// TIA Portal project "Mill3" (V17)

(* hardware
DEVICE "S7-1500/ET200MP station_1"  S7-1500 station
   slot 0: "Rail_0"  Rack  6ES7 590-1***0-0AA0
   slot 1: "PLC_1"  CPU 1512C-1 PN  6ES7 512-1CK01-0AB0  V2.9
      slot 3: "CPU display_1"  6ES7591-1AA00-0AA0
      slot 32768: "PROFINET interface_1"  X1
         slot 32769: "Port_1"  X1 P1
         slot 32770: "Port_2"  X1 P2
      slot 34817: "Virtual CP interface port_1"  Virtual CP interface port  Virtual CP interface port
*)

// ===== PLC "PLC_1"  CPU 1512C-1 PN =====

VAR_GLOBAL   // PLC tag table "Default tag table"
   "Tag_1" AT %M0.0 : Bool;
   "Tag_2" AT %M0.1 : Bool;
   "ResetPID" AT %I0.2 : Bool;
END_VAR

TYPE "Weigh_Feeder"
   STRUCT
      LoadCell_Reading : Real;
      Motor_Speed : Real;
      "SetPoint_%" : Real;
      SetPoint : Real;
      "Maximum_t/h" : Real;
   END_STRUCT;
END_TYPE

TYPE "Motors"
   STRUCT
      Start : Bool;
      Stop : Bool;
      "Motor_ON/OFF" : Bool;
   END_STRUCT;
END_TYPE

TYPE "Belts&BE"
   STRUCT
      Start : Bool;
      Stop : Bool;
      "Belt_ON/OFF" : Bool;
      BSS : Bool;
      PC : Bool;
      PC_Error : Bool;
      BSS_Error : Bool;
      Reset_Error : Bool;
   END_STRUCT;
END_TYPE

TYPE "Ratios"
   STRUCT
      Clinker : Real;
      Pozzolana : Real;
      Gypsum : Real;
      Limestone : Real;
      Select : Bool;
      Selected : Bool;
   END_STRUCT;
END_TYPE

TYPE "bagfilter"
   STRUCT
      Start : Bool;
      Stop : Bool;
      "On/Off" : Bool;
   END_STRUCT;
END_TYPE

TYPE "Reverse/Foward"
   STRUCT
      Foward : Bool;
      Reverse : Bool;
      Stop : Bool;
      PC : Bool;
      BSS : Bool;
      PC_Error : Bool;
      BSS_Error : Bool;
      Reset_Error : Bool;
      FWD_Mode : Bool;
      REV_Mode : Bool;
   END_STRUCT;
END_TYPE

// folder: DataBlocks

DATA_BLOCK "WeighFeeders(DB)"   // DB1
{ S7_Optimized_Access := 'TRUE' }
VERSION : 0.1
   VAR
      Pozzolana : "Weigh_Feeder";
      Clinker : "Weigh_Feeder";
      Gypsum : "Weigh_Feeder";
      Limestone : "Weigh_Feeder";
      Mill_TPH : Real := 310.0;
   END_VAR
BEGIN
   Pozzolana."Maximum_t/h" := 175.0;
   Clinker."Maximum_t/h" := 310.0;
   Gypsum."Maximum_t/h" := 35.0;
   Limestone."Maximum_t/h" := 75.0;
END_DATA_BLOCK

DATA_BLOCK "StartSystem"   // DB6
{ S7_Optimized_Access := 'TRUE' }
VERSION : 0.1
   VAR
      StartSystem : Bool;
      StopSystem : Bool;
      "Syste_ON/OFF" : Bool;
      Automatic_Selection : Bool;
      Manual_Selection : Bool;
      AuromaticMode : Bool;
      ManualMode : Bool;
      Siren : Bool;
      Main_BagFilter : "bagfilter";
      Mill_Drive : "Motors";
      "280KW FAN" : "Motors";
      MainBF_RotorAirLock : "Motors";
      Silo_Level : Int;
      Mill_Temp : Real := 23.0;
      level_Indication : Int;
      Timer1_PT : Time := T#15000ms;
      Timer2_PT : Time := T#10000ms;
   END_VAR
BEGIN
END_DATA_BLOCK

DATA_BLOCK "Belts|BE"   // DB9
{ S7_Optimized_Access := 'TRUE' }
VERSION : 0.1
   VAR
      Clinker : "Belts&BE";
      Pozzolana : "Belts&BE";
      Gypsum : "Belts&BE";
      Limestone : "Belts&BE";
      MaterialInlet_Belt : "Belts&BE";
      CourseMaterial_Belt : "Belts&BE";
      MillInlet_BE : "Belts&BE";
      OutletSilo_BE : "Belts&BE";
      FromYard_Belt : "Belts&BE";
      BF_To_OutletBE_Belt : "Belts&BE";
      "Clinker&Gypsum_Belt" : "Reverse/Foward";
      "Limestone&Pozzolana_Belt" : "Reverse/Foward";
   END_VAR
BEGIN
END_DATA_BLOCK

DATA_BLOCK "Material Rationing"   // DB10
{ S7_Optimized_Access := 'TRUE' }
VERSION : 0.1
   VAR
      Kp_Silver : "Ratios";
      Kp_Gold : "Ratios";
      Kp_Super_Gold : "Ratios";
      Kp_OPC : "Ratios";
   END_VAR
BEGIN
   Kp_Silver.Clinker := 52.0;
   Kp_Silver.Pozzolana := 40.0;
   Kp_Silver.Gypsum := 3.0;
   Kp_Silver.Limestone := 5.0;
   Kp_OPC.Clinker := 92.0;
   Kp_OPC.Pozzolana := 0.0;
   Kp_OPC.Gypsum := 5.0;
   Kp_OPC.Limestone := 3.0;
   Kp_Super_Gold.Clinker := 80.0;
   Kp_Super_Gold.Pozzolana := 10.0;
   Kp_Super_Gold.Gypsum := 5.0;
   Kp_Super_Gold.Limestone := 5.0;
   Kp_Gold.Clinker := 72.0;
   Kp_Gold.Pozzolana := 20.0;
   Kp_Gold.Gypsum := 5.0;
   Kp_Gold.Limestone := 3.0;
END_DATA_BLOCK

// folder: System blocks/Program resources

DATA_BLOCK "IEC_Timer_0_DB"   // DB7
{ S7_Optimized_Access := 'TRUE' }
AUTHOR : Simatic
FAMILY : IEC
NAME : IEC_TMR
VERSION : 1.0
// stored: InstanceOfName IEC_TIMER
"IEC_TIMER"
BEGIN
END_DATA_BLOCK

DATA_BLOCK "IEC_Timer_0_DB_1"   // DB8
{ S7_Optimized_Access := 'TRUE' }
AUTHOR : Simatic
FAMILY : IEC
NAME : IEC_TMR
VERSION : 1.0
// stored: InstanceOfName IEC_TIMER
"IEC_TIMER"
BEGIN
END_DATA_BLOCK

// folder: (top level)

ORGANIZATION_BLOCK "Main"   // OB1, LAD, ProgramCycle
TITLE = "Main Program Sweep (Cycle)"
{ S7_Optimized_Access := 'TRUE' }
VERSION : 0.1
   VAR_INPUT
      Initial_Call : Bool;   // Initial call of this OB
      Remanence : Bool;   // =True, if remanent data are available
   END_VAR
BEGIN

REGION Network 1: Start System Set| Stop System Reset
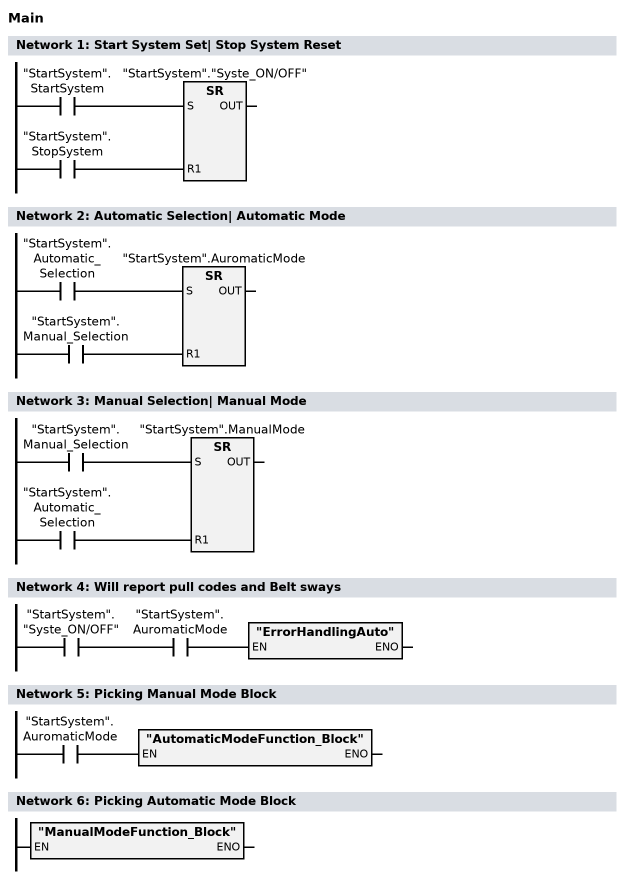
   RUNG wire#powerrail
      Contact( "StartSystem".StartSystem )
      S_SR(operand := "StartSystem"."Syste_ON/OFF", r1 := wire#w1)
   END_RUNG
   RUNG wire#powerrail
      Contact( "StartSystem".StopSystem )
   END_RUNG wire#w1
   // the same network as SCL:
   IF "StartSystem".StartSystem THEN
       "StartSystem"."Syste_ON/OFF" := TRUE;   // SR flip-flop
   END_IF;
   IF "StartSystem".StopSystem THEN "StartSystem"."Syste_ON/OFF" := FALSE; END_IF;
END_REGION

REGION Network 2: Automatic Selection| Automatic Mode
   RUNG wire#powerrail
      Contact( "StartSystem".Automatic_Selection )
      S_SR(operand := "StartSystem".AuromaticMode, r1 := wire#w1)
   END_RUNG
   RUNG wire#powerrail
      Contact( "StartSystem".Manual_Selection )
   END_RUNG wire#w1
   // the same network as SCL:
   IF "StartSystem".Automatic_Selection THEN
       "StartSystem".AuromaticMode := TRUE;   // SR flip-flop
   END_IF;
   IF "StartSystem".Manual_Selection THEN "StartSystem".AuromaticMode := FALSE; END_IF;
END_REGION

REGION Network 3: Manual Selection| Manual Mode
   RUNG wire#powerrail
      Contact( "StartSystem".Manual_Selection )
      S_SR(operand := "StartSystem".ManualMode, r1 := wire#w1)
   END_RUNG
   RUNG wire#powerrail
      Contact( "StartSystem".Automatic_Selection )
   END_RUNG wire#w1
   // the same network as SCL:
   IF "StartSystem".Manual_Selection THEN
       "StartSystem".ManualMode := TRUE;   // SR flip-flop
   END_IF;
   IF "StartSystem".Automatic_Selection THEN "StartSystem".ManualMode := FALSE; END_IF;
END_REGION

REGION Network 4: Will report pull codes and Belt sways
   RUNG wire#powerrail
      Contact( "StartSystem"."Syste_ON/OFF" )
      Contact( "StartSystem".AuromaticMode )
      "ErrorHandlingAuto"()
   END_RUNG
   // the same network as SCL:
   IF "StartSystem"."Syste_ON/OFF" AND "StartSystem".AuromaticMode THEN "ErrorHandlingAuto"(); END_IF;
END_REGION

REGION Network 5: Picking Manual Mode Block
   RUNG wire#powerrail
      Contact( "StartSystem".AuromaticMode )
      "AutomaticModeFunction_Block"()
   END_RUNG
   // the same network as SCL:
   IF "StartSystem".AuromaticMode THEN "AutomaticModeFunction_Block"(); END_IF;
END_REGION

REGION Network 6: Picking Automatic Mode Block
   RUNG wire#powerrail
      "ManualModeFunction_Block"()
   END_RUNG
   // the same network as SCL:
   "ManualModeFunction_Block"();
END_REGION
END_ORGANIZATION_BLOCK

ORGANIZATION_BLOCK "Cyclic interrupt_Level&Temp Simulation"   // OB32, LAD, CyclicInterrupt
{ S7_Optimized_Access := 'TRUE' }
VERSION : 0.1
   VAR_INPUT
      Initial_Call : Bool;   // Initial call of this OB
      Event_Count : Int;   // Events discarded
   END_VAR
   VAR_TEMP
      CalcOut : Real;
      level_Out : Real;
   END_VAR
BEGIN

REGION Network 1: Mill Temperature Increasing while first timer 1 is timing
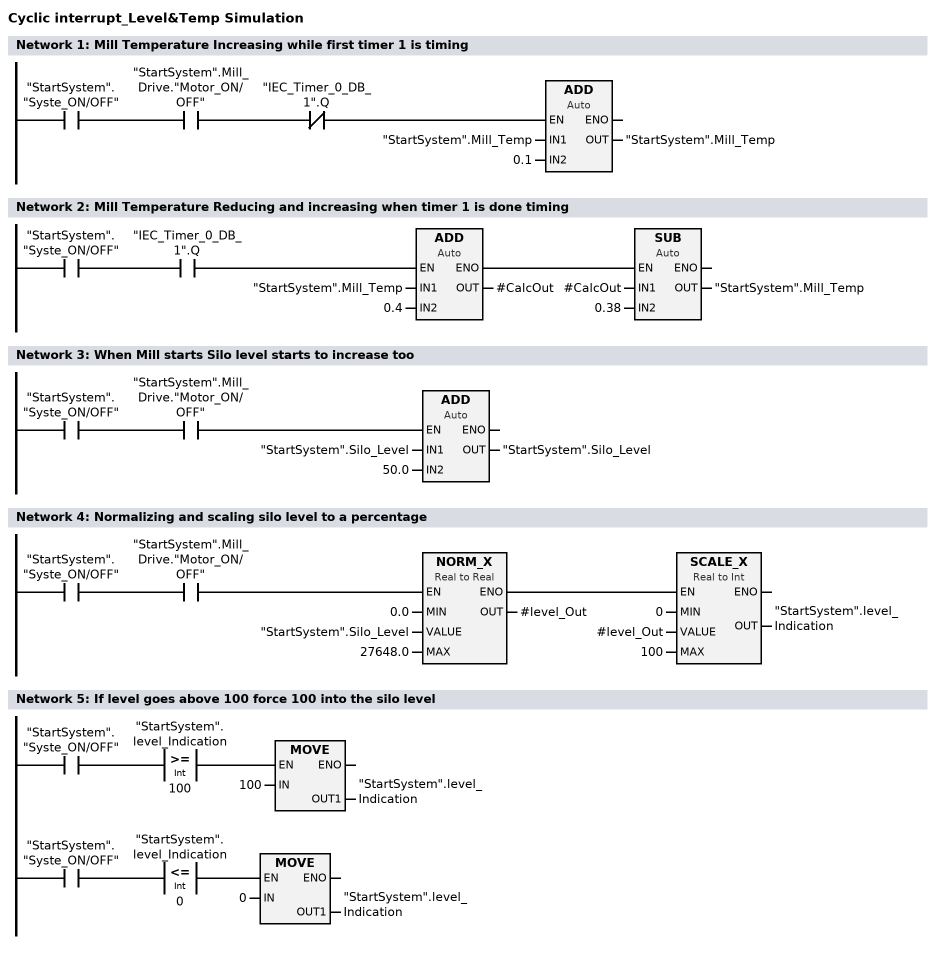
   RUNG wire#powerrail
      Contact( "StartSystem"."Syste_ON/OFF" )
      Contact( "StartSystem".Mill_Drive."Motor_ON/OFF" )
      I_Contact( "IEC_Timer_0_DB_1".Q )
      Add(in1 := "StartSystem".Mill_Temp, in2 := 0.1, out => "StartSystem".Mill_Temp)
   END_RUNG
   // the same network as SCL:
   IF "StartSystem"."Syste_ON/OFF" AND "StartSystem".Mill_Drive."Motor_ON/OFF" AND NOT "IEC_Timer_0_DB_1".Q THEN
       "StartSystem".Mill_Temp := "StartSystem".Mill_Temp + 0.1;
   END_IF;
END_REGION

REGION Network 2: Mill Temperature Reducing and increasing when timer 1 is done timing
   RUNG wire#powerrail
      Contact( "StartSystem"."Syste_ON/OFF" )
      Contact( "IEC_Timer_0_DB_1".Q )
      Add(in1 := "StartSystem".Mill_Temp, in2 := 0.4, out => #CalcOut)
      Sub(in1 := #CalcOut, in2 := 0.38, out => "StartSystem".Mill_Temp)
   END_RUNG
   // the same network as SCL:
   IF "StartSystem"."Syste_ON/OFF" AND "IEC_Timer_0_DB_1".Q THEN
       #CalcOut := "StartSystem".Mill_Temp + 0.4;
       "StartSystem".Mill_Temp := #CalcOut - 0.38;
   END_IF;
END_REGION

REGION Network 3: When Mill starts Silo level starts to increase too
   RUNG wire#powerrail
      Contact( "StartSystem"."Syste_ON/OFF" )
      Contact( "StartSystem".Mill_Drive."Motor_ON/OFF" )
      Add(in1 := "StartSystem".Silo_Level, in2 := 50.0, out => "StartSystem".Silo_Level)
   END_RUNG
   // the same network as SCL:
   IF "StartSystem"."Syste_ON/OFF" AND "StartSystem".Mill_Drive."Motor_ON/OFF" THEN
       "StartSystem".Silo_Level := "StartSystem".Silo_Level + 50.0;
   END_IF;
END_REGION

REGION Network 4: Normalizing and scaling silo level to a percentage
   RUNG wire#powerrail
      Contact( "StartSystem"."Syste_ON/OFF" )
      Contact( "StartSystem".Mill_Drive."Motor_ON/OFF" )
      { S7_Templates := "[SrcType := Real, DestType := Real]" } Normalize(min := 0.0, value := "StartSystem".Silo_Level, max := 27648.0, out => #level_Out)
      { S7_Templates := "[SrcType := Real, DestType := Int]" } Scale(min := 0, value := #level_Out, max := 100, out => "StartSystem".level_Indication)
   END_RUNG
   // the same network as SCL:
   IF "StartSystem"."Syste_ON/OFF" AND "StartSystem".Mill_Drive."Motor_ON/OFF" THEN
       #level_Out := NORM_X(MIN := 0.0, VALUE := "StartSystem".Silo_Level, MAX := 27648.0);
       "StartSystem".level_Indication := SCALE_X(MIN := 0, VALUE := #level_Out, MAX := 100);
   END_IF;
END_REGION

REGION Network 5: If level goes above 100 force 100 into the silo level
   RUNG wire#powerrail
      Contact( "StartSystem"."Syste_ON/OFF" )
      { S7_Templates := "SrcType := Int" } GE_Contact(in1 := "StartSystem".level_Indication, in2 := 100)
      Move(in := 100, out1 => "StartSystem".level_Indication)
   END_RUNG
   RUNG wire#powerrail
      Contact( "StartSystem"."Syste_ON/OFF" )
      { S7_Templates := "SrcType := Int" } LE_Contact(in1 := "StartSystem".level_Indication, in2 := 0)
      Move(in := 0, out1 => "StartSystem".level_Indication)
   END_RUNG
   // the same network as SCL:
   IF "StartSystem"."Syste_ON/OFF" AND ("StartSystem".level_Indication >= 100) THEN
       "StartSystem".level_Indication := 100;
   END_IF;
   IF "StartSystem"."Syste_ON/OFF" AND ("StartSystem".level_Indication <= 0) THEN
       "StartSystem".level_Indication := 0;
   END_IF;
END_REGION
END_ORGANIZATION_BLOCK

// folder: Auto_Mode

FUNCTION "AutomaticModeFunction_Block" : Void   // FC5, LAD
{ S7_Optimized_Access := 'TRUE' }
VERSION : 0.1
   VAR_TEMP   // added for the SCL form of the ladder/FBD networks
      _w1 : Bool;
   END_VAR
BEGIN

REGION Network 1: Main FAN, Main Bag Filter and Main Bag Filter rotor airlock goes on
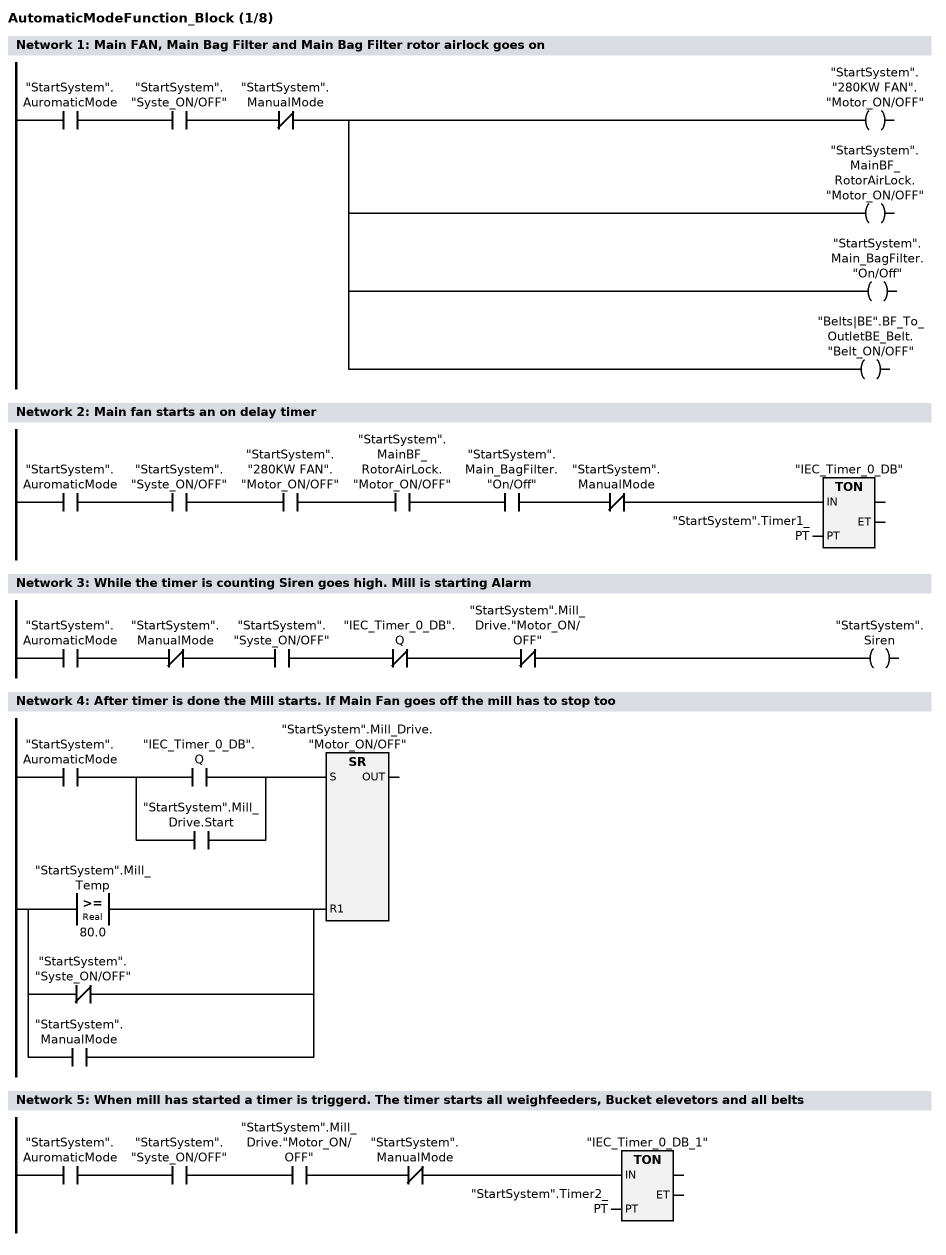
   RUNG wire#powerrail
      Contact( "StartSystem".AuromaticMode )
      Contact( "StartSystem"."Syste_ON/OFF" )
      I_Contact( "StartSystem".ManualMode )
      wire#w1
      Coil( "StartSystem"."280KW FAN"."Motor_ON/OFF" )
   END_RUNG
   RUNG wire#w1
      Coil( "StartSystem".MainBF_RotorAirLock."Motor_ON/OFF" )
   END_RUNG
   RUNG wire#w1
      Coil( "StartSystem".Main_BagFilter."On/Off" )
   END_RUNG
   RUNG wire#w1
      Coil( "Belts|BE".BF_To_OutletBE_Belt."Belt_ON/OFF" )
   END_RUNG
   // the same network as SCL:
   "StartSystem"."280KW FAN"."Motor_ON/OFF" := "StartSystem".AuromaticMode AND "StartSystem"."Syste_ON/OFF" AND NOT "StartSystem".ManualMode;
   "StartSystem".MainBF_RotorAirLock."Motor_ON/OFF" := "StartSystem"."280KW FAN"."Motor_ON/OFF";
   "StartSystem".Main_BagFilter."On/Off" := "StartSystem"."280KW FAN"."Motor_ON/OFF";
   "Belts|BE".BF_To_OutletBE_Belt."Belt_ON/OFF" := "StartSystem"."280KW FAN"."Motor_ON/OFF";
END_REGION

REGION Network 2: Main fan starts an on delay timer
   "IEC_Timer_0_DB".TON(IN := "StartSystem".AuromaticMode AND "StartSystem"."Syste_ON/OFF" AND "StartSystem"."280KW FAN"."Motor_ON/OFF" AND "StartSystem".MainBF_RotorAirLock."Motor_ON/OFF" AND "StartSystem".Main_BagFilter."On/Off" AND NOT "StartSystem".ManualMode,
                        PT := "StartSystem".Timer1_PT);
END_REGION

REGION Network 3: While the timer is counting Siren goes high. Mill is starting Alarm
   RUNG wire#powerrail
      Contact( "StartSystem".AuromaticMode )
      I_Contact( "StartSystem".ManualMode )
      Contact( "StartSystem"."Syste_ON/OFF" )
      I_Contact( "IEC_Timer_0_DB".Q )
      I_Contact( "StartSystem".Mill_Drive."Motor_ON/OFF" )
      Coil( "StartSystem".Siren )
   END_RUNG
   // the same network as SCL:
   "StartSystem".Siren := "StartSystem".AuromaticMode AND NOT "StartSystem".ManualMode AND "StartSystem"."Syste_ON/OFF" AND NOT "IEC_Timer_0_DB".Q AND NOT "StartSystem".Mill_Drive."Motor_ON/OFF";
END_REGION

REGION Network 4: After timer is done the Mill starts. If Main Fan goes off the mill has to stop too
   RUNG wire#powerrail
      Contact( "StartSystem".AuromaticMode )
      wire#w1
      Contact( "IEC_Timer_0_DB".Q )
      wire#w2
      S_SR(operand := "StartSystem".Mill_Drive."Motor_ON/OFF", r1 := wire#w3)
   END_RUNG
   RUNG wire#w1
      Contact( "StartSystem".Mill_Drive.Start )
   END_RUNG wire#w2
   RUNG wire#powerrail
      { S7_Templates := "SrcType := Real" } GE_Contact(in1 := "StartSystem".Mill_Temp, in2 := 80.0)
   END_RUNG wire#w3
   RUNG wire#powerrail
      I_Contact( "StartSystem"."Syste_ON/OFF" )
   END_RUNG wire#w3
   RUNG wire#powerrail
      Contact( "StartSystem".ManualMode )
   END_RUNG wire#w3
   // the same network as SCL:
   IF "StartSystem".AuromaticMode AND ("IEC_Timer_0_DB".Q OR "StartSystem".Mill_Drive.Start) THEN
       "StartSystem".Mill_Drive."Motor_ON/OFF" := TRUE;   // SR flip-flop
   END_IF;
   IF ("StartSystem".Mill_Temp >= 80.0) OR NOT "StartSystem"."Syste_ON/OFF" OR "StartSystem".ManualMode THEN
       "StartSystem".Mill_Drive."Motor_ON/OFF" := FALSE;
   END_IF;
END_REGION

REGION Network 5: When mill has started a timer is triggerd. The timer starts all weighfeeders, Bucket elevetors and all belts
   "IEC_Timer_0_DB_1".TON(IN := "StartSystem".AuromaticMode AND "StartSystem"."Syste_ON/OFF" AND "StartSystem".Mill_Drive."Motor_ON/OFF" AND NOT "StartSystem".ManualMode,
                          PT := "StartSystem".Timer2_PT);
END_REGION

REGION Network 6: Starting Clinker WF Belt
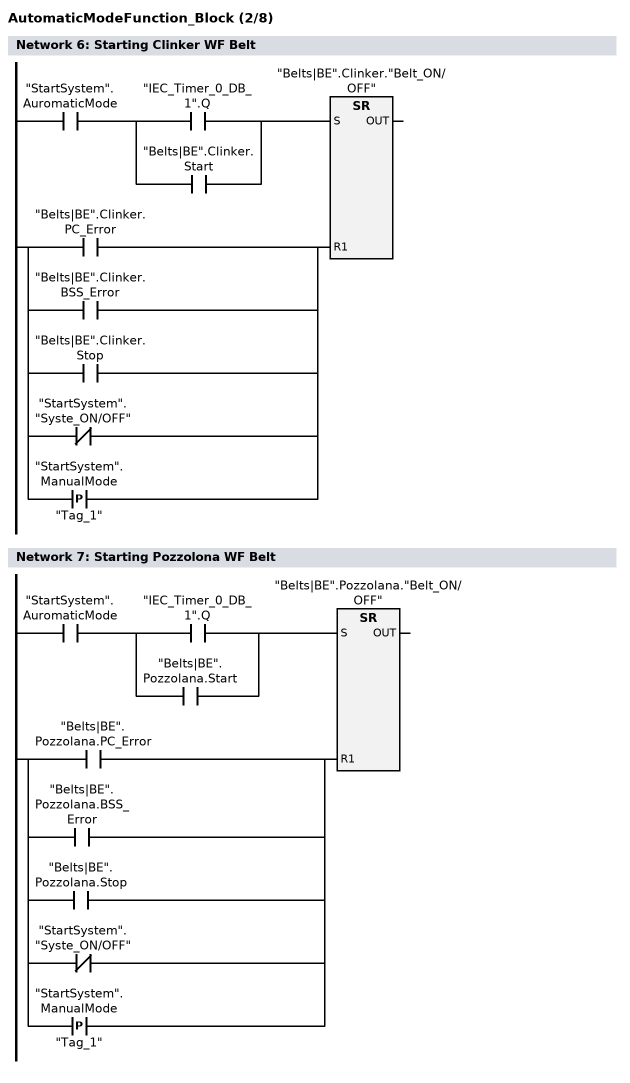
   RUNG wire#powerrail
      Contact( "StartSystem".AuromaticMode )
      wire#w1
      Contact( "IEC_Timer_0_DB_1".Q )
      wire#w2
      S_SR(operand := "Belts|BE".Clinker."Belt_ON/OFF", r1 := wire#w3)
   END_RUNG
   RUNG wire#w1
      Contact( "Belts|BE".Clinker.Start )
   END_RUNG wire#w2
   RUNG wire#powerrail
      Contact( "Belts|BE".Clinker.PC_Error )
   END_RUNG wire#w3
   RUNG wire#powerrail
      Contact( "Belts|BE".Clinker.BSS_Error )
   END_RUNG wire#w3
   RUNG wire#powerrail
      Contact( "Belts|BE".Clinker.Stop )
   END_RUNG wire#w3
   RUNG wire#powerrail
      I_Contact( "StartSystem"."Syste_ON/OFF" )
   END_RUNG wire#w3
   RUNG wire#powerrail
      P_Contact(operand := "StartSystem".ManualMode, bit := "Tag_1")
   END_RUNG wire#w3
   // the same network as SCL:
   #_w1 := "StartSystem".ManualMode AND NOT "Tag_1";   // rising edge of "StartSystem".ManualMode
   "Tag_1" := "StartSystem".ManualMode;
   IF "StartSystem".AuromaticMode AND ("IEC_Timer_0_DB_1".Q OR "Belts|BE".Clinker.Start) THEN
       "Belts|BE".Clinker."Belt_ON/OFF" := TRUE;   // SR flip-flop
   END_IF;
   IF "Belts|BE".Clinker.PC_Error OR "Belts|BE".Clinker.BSS_Error OR "Belts|BE".Clinker.Stop OR NOT "StartSystem"."Syste_ON/OFF" OR #_w1 THEN
       "Belts|BE".Clinker."Belt_ON/OFF" := FALSE;
   END_IF;
END_REGION

REGION Network 7: Starting Pozzolona WF Belt
   RUNG wire#powerrail
      Contact( "StartSystem".AuromaticMode )
      wire#w1
      Contact( "IEC_Timer_0_DB_1".Q )
      wire#w2
      S_SR(operand := "Belts|BE".Pozzolana."Belt_ON/OFF", r1 := wire#w3)
   END_RUNG
   RUNG wire#w1
      Contact( "Belts|BE".Pozzolana.Start )
   END_RUNG wire#w2
   RUNG wire#powerrail
      Contact( "Belts|BE".Pozzolana.PC_Error )
   END_RUNG wire#w3
   RUNG wire#powerrail
      Contact( "Belts|BE".Pozzolana.BSS_Error )
   END_RUNG wire#w3
   RUNG wire#powerrail
      Contact( "Belts|BE".Pozzolana.Stop )
   END_RUNG wire#w3
   RUNG wire#powerrail
      I_Contact( "StartSystem"."Syste_ON/OFF" )
   END_RUNG wire#w3
   RUNG wire#powerrail
      P_Contact(operand := "StartSystem".ManualMode, bit := "Tag_1")
   END_RUNG wire#w3
   // the same network as SCL:
   #_w1 := "StartSystem".ManualMode AND NOT "Tag_1";   // rising edge of "StartSystem".ManualMode
   "Tag_1" := "StartSystem".ManualMode;
   IF "StartSystem".AuromaticMode AND ("IEC_Timer_0_DB_1".Q OR "Belts|BE".Pozzolana.Start) THEN
       "Belts|BE".Pozzolana."Belt_ON/OFF" := TRUE;   // SR flip-flop
   END_IF;
   IF "Belts|BE".Pozzolana.PC_Error OR "Belts|BE".Pozzolana.BSS_Error OR "Belts|BE".Pozzolana.Stop OR NOT "StartSystem"."Syste_ON/OFF" OR #_w1 THEN
       "Belts|BE".Pozzolana."Belt_ON/OFF" := FALSE;
   END_IF;
END_REGION

REGION Network 8: Starting Gypsum WF Belt
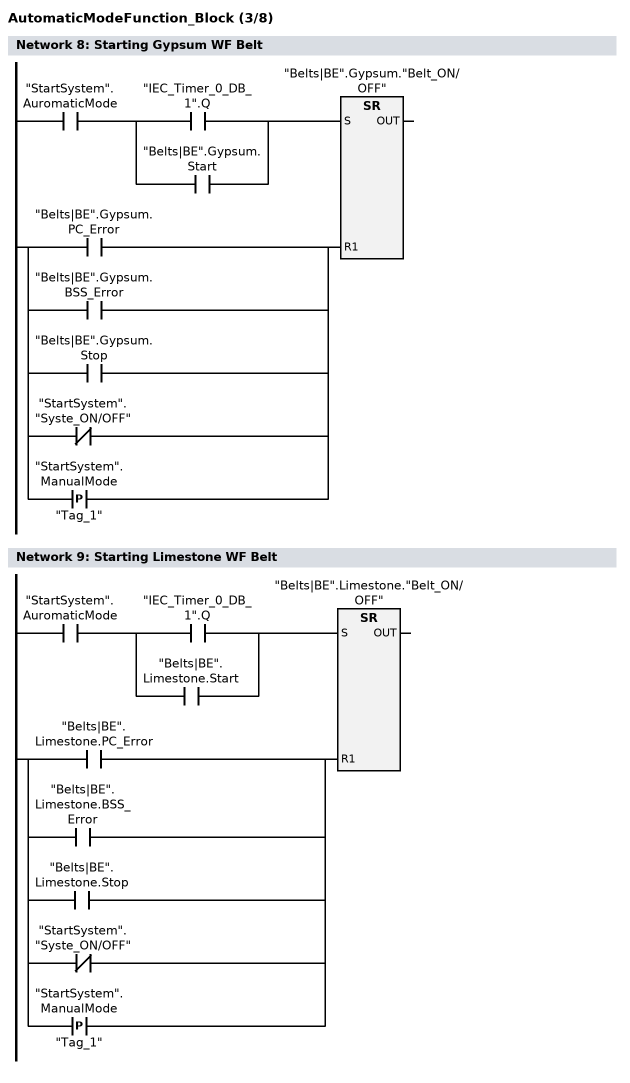
   RUNG wire#powerrail
      Contact( "StartSystem".AuromaticMode )
      wire#w1
      Contact( "IEC_Timer_0_DB_1".Q )
      wire#w2
      S_SR(operand := "Belts|BE".Gypsum."Belt_ON/OFF", r1 := wire#w3)
   END_RUNG
   RUNG wire#w1
      Contact( "Belts|BE".Gypsum.Start )
   END_RUNG wire#w2
   RUNG wire#powerrail
      Contact( "Belts|BE".Gypsum.PC_Error )
   END_RUNG wire#w3
   RUNG wire#powerrail
      Contact( "Belts|BE".Gypsum.BSS_Error )
   END_RUNG wire#w3
   RUNG wire#powerrail
      Contact( "Belts|BE".Gypsum.Stop )
   END_RUNG wire#w3
   RUNG wire#powerrail
      I_Contact( "StartSystem"."Syste_ON/OFF" )
   END_RUNG wire#w3
   RUNG wire#powerrail
      P_Contact(operand := "StartSystem".ManualMode, bit := "Tag_1")
   END_RUNG wire#w3
   // the same network as SCL:
   #_w1 := "StartSystem".ManualMode AND NOT "Tag_1";   // rising edge of "StartSystem".ManualMode
   "Tag_1" := "StartSystem".ManualMode;
   IF "StartSystem".AuromaticMode AND ("IEC_Timer_0_DB_1".Q OR "Belts|BE".Gypsum.Start) THEN
       "Belts|BE".Gypsum."Belt_ON/OFF" := TRUE;   // SR flip-flop
   END_IF;
   IF "Belts|BE".Gypsum.PC_Error OR "Belts|BE".Gypsum.BSS_Error OR "Belts|BE".Gypsum.Stop OR NOT "StartSystem"."Syste_ON/OFF" OR #_w1 THEN
       "Belts|BE".Gypsum."Belt_ON/OFF" := FALSE;
   END_IF;
END_REGION

REGION Network 9: Starting Limestone WF Belt
   RUNG wire#powerrail
      Contact( "StartSystem".AuromaticMode )
      wire#w1
      Contact( "IEC_Timer_0_DB_1".Q )
      wire#w2
      S_SR(operand := "Belts|BE".Limestone."Belt_ON/OFF", r1 := wire#w3)
   END_RUNG
   RUNG wire#w1
      Contact( "Belts|BE".Limestone.Start )
   END_RUNG wire#w2
   RUNG wire#powerrail
      Contact( "Belts|BE".Limestone.PC_Error )
   END_RUNG wire#w3
   RUNG wire#powerrail
      Contact( "Belts|BE".Limestone.BSS_Error )
   END_RUNG wire#w3
   RUNG wire#powerrail
      Contact( "Belts|BE".Limestone.Stop )
   END_RUNG wire#w3
   RUNG wire#powerrail
      I_Contact( "StartSystem"."Syste_ON/OFF" )
   END_RUNG wire#w3
   RUNG wire#powerrail
      P_Contact(operand := "StartSystem".ManualMode, bit := "Tag_1")
   END_RUNG wire#w3
   // the same network as SCL:
   #_w1 := "StartSystem".ManualMode AND NOT "Tag_1";   // rising edge of "StartSystem".ManualMode
   "Tag_1" := "StartSystem".ManualMode;
   IF "StartSystem".AuromaticMode AND ("IEC_Timer_0_DB_1".Q OR "Belts|BE".Limestone.Start) THEN
       "Belts|BE".Limestone."Belt_ON/OFF" := TRUE;   // SR flip-flop
   END_IF;
   IF "Belts|BE".Limestone.PC_Error OR "Belts|BE".Limestone.BSS_Error OR "Belts|BE".Limestone.Stop OR NOT "StartSystem"."Syste_ON/OFF" OR #_w1 THEN
       "Belts|BE".Limestone."Belt_ON/OFF" := FALSE;
   END_IF;
END_REGION

REGION Network 10: Starting Material Inlet Long Belts. If belts sways or pull code is activated specific belts go off untill reset
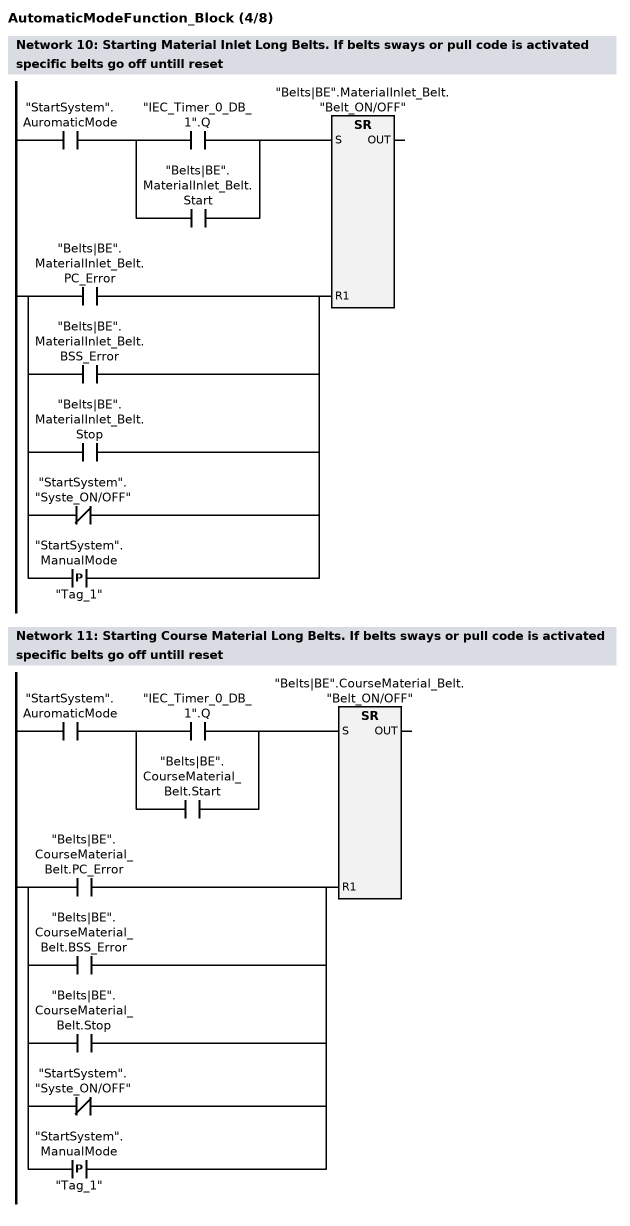
   RUNG wire#powerrail
      Contact( "StartSystem".AuromaticMode )
      wire#w1
      Contact( "IEC_Timer_0_DB_1".Q )
      wire#w2
      S_SR(operand := "Belts|BE".MaterialInlet_Belt."Belt_ON/OFF", r1 := wire#w3)
   END_RUNG
   RUNG wire#w1
      Contact( "Belts|BE".MaterialInlet_Belt.Start )
   END_RUNG wire#w2
   RUNG wire#powerrail
      Contact( "Belts|BE".MaterialInlet_Belt.PC_Error )
   END_RUNG wire#w3
   RUNG wire#powerrail
      Contact( "Belts|BE".MaterialInlet_Belt.BSS_Error )
   END_RUNG wire#w3
   RUNG wire#powerrail
      Contact( "Belts|BE".MaterialInlet_Belt.Stop )
   END_RUNG wire#w3
   RUNG wire#powerrail
      I_Contact( "StartSystem"."Syste_ON/OFF" )
   END_RUNG wire#w3
   RUNG wire#powerrail
      P_Contact(operand := "StartSystem".ManualMode, bit := "Tag_1")
   END_RUNG wire#w3
   // the same network as SCL:
   #_w1 := "StartSystem".ManualMode AND NOT "Tag_1";   // rising edge of "StartSystem".ManualMode
   "Tag_1" := "StartSystem".ManualMode;
   IF "StartSystem".AuromaticMode AND ("IEC_Timer_0_DB_1".Q OR "Belts|BE".MaterialInlet_Belt.Start) THEN
       "Belts|BE".MaterialInlet_Belt."Belt_ON/OFF" := TRUE;   // SR flip-flop
   END_IF;
   IF "Belts|BE".MaterialInlet_Belt.PC_Error OR "Belts|BE".MaterialInlet_Belt.BSS_Error OR "Belts|BE".MaterialInlet_Belt.Stop OR NOT "StartSystem"."Syste_ON/OFF" OR #_w1 THEN
       "Belts|BE".MaterialInlet_Belt."Belt_ON/OFF" := FALSE;
   END_IF;
END_REGION

REGION Network 11: Starting Course Material Long Belts. If belts sways or pull code is activated specific belts go off untill reset
   RUNG wire#powerrail
      Contact( "StartSystem".AuromaticMode )
      wire#w1
      Contact( "IEC_Timer_0_DB_1".Q )
      wire#w2
      S_SR(operand := "Belts|BE".CourseMaterial_Belt."Belt_ON/OFF", r1 := wire#w3)
   END_RUNG
   RUNG wire#w1
      Contact( "Belts|BE".CourseMaterial_Belt.Start )
   END_RUNG wire#w2
   RUNG wire#powerrail
      Contact( "Belts|BE".CourseMaterial_Belt.PC_Error )
   END_RUNG wire#w3
   RUNG wire#powerrail
      Contact( "Belts|BE".CourseMaterial_Belt.BSS_Error )
   END_RUNG wire#w3
   RUNG wire#powerrail
      Contact( "Belts|BE".CourseMaterial_Belt.Stop )
   END_RUNG wire#w3
   RUNG wire#powerrail
      I_Contact( "StartSystem"."Syste_ON/OFF" )
   END_RUNG wire#w3
   RUNG wire#powerrail
      P_Contact(operand := "StartSystem".ManualMode, bit := "Tag_1")
   END_RUNG wire#w3
   // the same network as SCL:
   #_w1 := "StartSystem".ManualMode AND NOT "Tag_1";   // rising edge of "StartSystem".ManualMode
   "Tag_1" := "StartSystem".ManualMode;
   IF "StartSystem".AuromaticMode AND ("IEC_Timer_0_DB_1".Q OR "Belts|BE".CourseMaterial_Belt.Start) THEN
       "Belts|BE".CourseMaterial_Belt."Belt_ON/OFF" := TRUE;   // SR flip-flop
   END_IF;
   IF "Belts|BE".CourseMaterial_Belt.PC_Error OR "Belts|BE".CourseMaterial_Belt.BSS_Error OR "Belts|BE".CourseMaterial_Belt.Stop OR NOT "StartSystem"."Syste_ON/OFF" OR #_w1 THEN
       "Belts|BE".CourseMaterial_Belt."Belt_ON/OFF" := FALSE;
   END_IF;
END_REGION

REGION Network 12: Starting Inlet Bucket Elevetor. If belts sways or pull code is activated specific belts go off untill reset
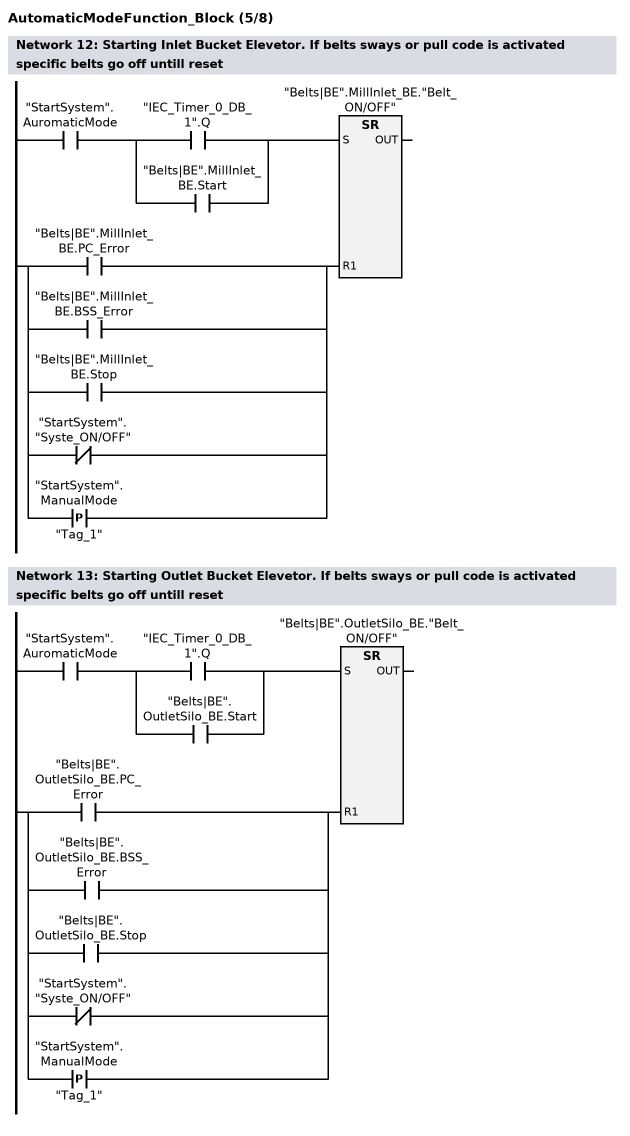
   RUNG wire#powerrail
      Contact( "StartSystem".AuromaticMode )
      wire#w1
      Contact( "IEC_Timer_0_DB_1".Q )
      wire#w2
      S_SR(operand := "Belts|BE".MillInlet_BE."Belt_ON/OFF", r1 := wire#w3)
   END_RUNG
   RUNG wire#w1
      Contact( "Belts|BE".MillInlet_BE.Start )
   END_RUNG wire#w2
   RUNG wire#powerrail
      Contact( "Belts|BE".MillInlet_BE.PC_Error )
   END_RUNG wire#w3
   RUNG wire#powerrail
      Contact( "Belts|BE".MillInlet_BE.BSS_Error )
   END_RUNG wire#w3
   RUNG wire#powerrail
      Contact( "Belts|BE".MillInlet_BE.Stop )
   END_RUNG wire#w3
   RUNG wire#powerrail
      I_Contact( "StartSystem"."Syste_ON/OFF" )
   END_RUNG wire#w3
   RUNG wire#powerrail
      P_Contact(operand := "StartSystem".ManualMode, bit := "Tag_1")
   END_RUNG wire#w3
   // the same network as SCL:
   #_w1 := "StartSystem".ManualMode AND NOT "Tag_1";   // rising edge of "StartSystem".ManualMode
   "Tag_1" := "StartSystem".ManualMode;
   IF "StartSystem".AuromaticMode AND ("IEC_Timer_0_DB_1".Q OR "Belts|BE".MillInlet_BE.Start) THEN
       "Belts|BE".MillInlet_BE."Belt_ON/OFF" := TRUE;   // SR flip-flop
   END_IF;
   IF "Belts|BE".MillInlet_BE.PC_Error OR "Belts|BE".MillInlet_BE.BSS_Error OR "Belts|BE".MillInlet_BE.Stop OR NOT "StartSystem"."Syste_ON/OFF" OR #_w1 THEN
       "Belts|BE".MillInlet_BE."Belt_ON/OFF" := FALSE;
   END_IF;
END_REGION

REGION Network 13: Starting Outlet Bucket Elevetor. If belts sways or pull code is activated specific belts go off untill reset
   RUNG wire#powerrail
      Contact( "StartSystem".AuromaticMode )
      wire#w1
      Contact( "IEC_Timer_0_DB_1".Q )
      wire#w2
      S_SR(operand := "Belts|BE".OutletSilo_BE."Belt_ON/OFF", r1 := wire#w3)
   END_RUNG
   RUNG wire#w1
      Contact( "Belts|BE".OutletSilo_BE.Start )
   END_RUNG wire#w2
   RUNG wire#powerrail
      Contact( "Belts|BE".OutletSilo_BE.PC_Error )
   END_RUNG wire#w3
   RUNG wire#powerrail
      Contact( "Belts|BE".OutletSilo_BE.BSS_Error )
   END_RUNG wire#w3
   RUNG wire#powerrail
      Contact( "Belts|BE".OutletSilo_BE.Stop )
   END_RUNG wire#w3
   RUNG wire#powerrail
      I_Contact( "StartSystem"."Syste_ON/OFF" )
   END_RUNG wire#w3
   RUNG wire#powerrail
      P_Contact(operand := "StartSystem".ManualMode, bit := "Tag_1")
   END_RUNG wire#w3
   // the same network as SCL:
   #_w1 := "StartSystem".ManualMode AND NOT "Tag_1";   // rising edge of "StartSystem".ManualMode
   "Tag_1" := "StartSystem".ManualMode;
   IF "StartSystem".AuromaticMode AND ("IEC_Timer_0_DB_1".Q OR "Belts|BE".OutletSilo_BE.Start) THEN
       "Belts|BE".OutletSilo_BE."Belt_ON/OFF" := TRUE;   // SR flip-flop
   END_IF;
   IF "Belts|BE".OutletSilo_BE.PC_Error OR "Belts|BE".OutletSilo_BE.BSS_Error OR "Belts|BE".OutletSilo_BE.Stop OR NOT "StartSystem"."Syste_ON/OFF" OR #_w1 THEN
       "Belts|BE".OutletSilo_BE."Belt_ON/OFF" := FALSE;
   END_IF;
END_REGION

REGION Network 14: Starting Belt From Material Yard to hoppers. If belts sways or pull code is activated specific belts go off untill reset
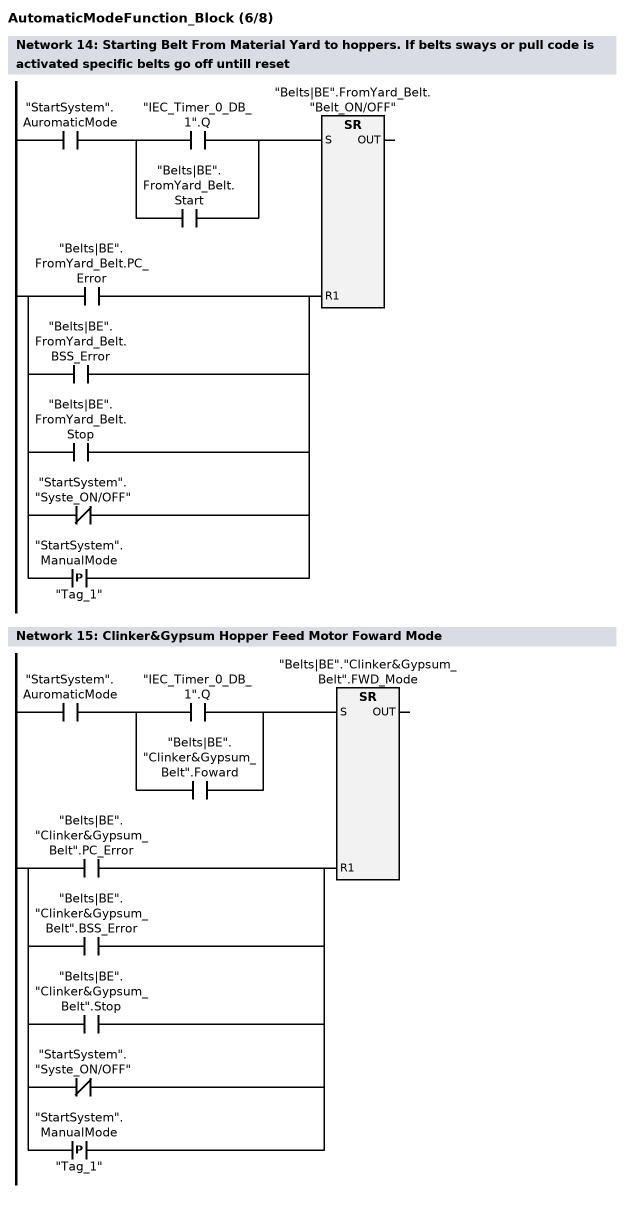
   RUNG wire#powerrail
      Contact( "StartSystem".AuromaticMode )
      wire#w1
      Contact( "IEC_Timer_0_DB_1".Q )
      wire#w2
      S_SR(operand := "Belts|BE".FromYard_Belt."Belt_ON/OFF", r1 := wire#w3)
   END_RUNG
   RUNG wire#w1
      Contact( "Belts|BE".FromYard_Belt.Start )
   END_RUNG wire#w2
   RUNG wire#powerrail
      Contact( "Belts|BE".FromYard_Belt.PC_Error )
   END_RUNG wire#w3
   RUNG wire#powerrail
      Contact( "Belts|BE".FromYard_Belt.BSS_Error )
   END_RUNG wire#w3
   RUNG wire#powerrail
      Contact( "Belts|BE".FromYard_Belt.Stop )
   END_RUNG wire#w3
   RUNG wire#powerrail
      I_Contact( "StartSystem"."Syste_ON/OFF" )
   END_RUNG wire#w3
   RUNG wire#powerrail
      P_Contact(operand := "StartSystem".ManualMode, bit := "Tag_1")
   END_RUNG wire#w3
   // the same network as SCL:
   #_w1 := "StartSystem".ManualMode AND NOT "Tag_1";   // rising edge of "StartSystem".ManualMode
   "Tag_1" := "StartSystem".ManualMode;
   IF "StartSystem".AuromaticMode AND ("IEC_Timer_0_DB_1".Q OR "Belts|BE".FromYard_Belt.Start) THEN
       "Belts|BE".FromYard_Belt."Belt_ON/OFF" := TRUE;   // SR flip-flop
   END_IF;
   IF "Belts|BE".FromYard_Belt.PC_Error OR "Belts|BE".FromYard_Belt.BSS_Error OR "Belts|BE".FromYard_Belt.Stop OR NOT "StartSystem"."Syste_ON/OFF" OR #_w1 THEN
       "Belts|BE".FromYard_Belt."Belt_ON/OFF" := FALSE;
   END_IF;
END_REGION

REGION Network 15: Clinker&Gypsum Hopper Feed Motor Foward Mode
   RUNG wire#powerrail
      Contact( "StartSystem".AuromaticMode )
      wire#w1
      Contact( "IEC_Timer_0_DB_1".Q )
      wire#w2
      S_SR(operand := "Belts|BE"."Clinker&Gypsum_Belt".FWD_Mode, r1 := wire#w3)
   END_RUNG
   RUNG wire#w1
      Contact( "Belts|BE"."Clinker&Gypsum_Belt".Foward )
   END_RUNG wire#w2
   RUNG wire#powerrail
      Contact( "Belts|BE"."Clinker&Gypsum_Belt".PC_Error )
   END_RUNG wire#w3
   RUNG wire#powerrail
      Contact( "Belts|BE"."Clinker&Gypsum_Belt".BSS_Error )
   END_RUNG wire#w3
   RUNG wire#powerrail
      Contact( "Belts|BE"."Clinker&Gypsum_Belt".Stop )
   END_RUNG wire#w3
   RUNG wire#powerrail
      I_Contact( "StartSystem"."Syste_ON/OFF" )
   END_RUNG wire#w3
   RUNG wire#powerrail
      P_Contact(operand := "StartSystem".ManualMode, bit := "Tag_1")
   END_RUNG wire#w3
   // the same network as SCL:
   #_w1 := "StartSystem".ManualMode AND NOT "Tag_1";   // rising edge of "StartSystem".ManualMode
   "Tag_1" := "StartSystem".ManualMode;
   IF "StartSystem".AuromaticMode AND ("IEC_Timer_0_DB_1".Q OR "Belts|BE"."Clinker&Gypsum_Belt".Foward) THEN
       "Belts|BE"."Clinker&Gypsum_Belt".FWD_Mode := TRUE;   // SR flip-flop
   END_IF;
   IF "Belts|BE"."Clinker&Gypsum_Belt".PC_Error OR "Belts|BE"."Clinker&Gypsum_Belt".BSS_Error OR "Belts|BE"."Clinker&Gypsum_Belt".Stop OR NOT "StartSystem"."Syste_ON/OFF" OR #_w1 THEN
       "Belts|BE"."Clinker&Gypsum_Belt".FWD_Mode := FALSE;
   END_IF;
END_REGION

REGION Network 16: Clinker&Gypsum Hopper Feed Motor Reverse Mode
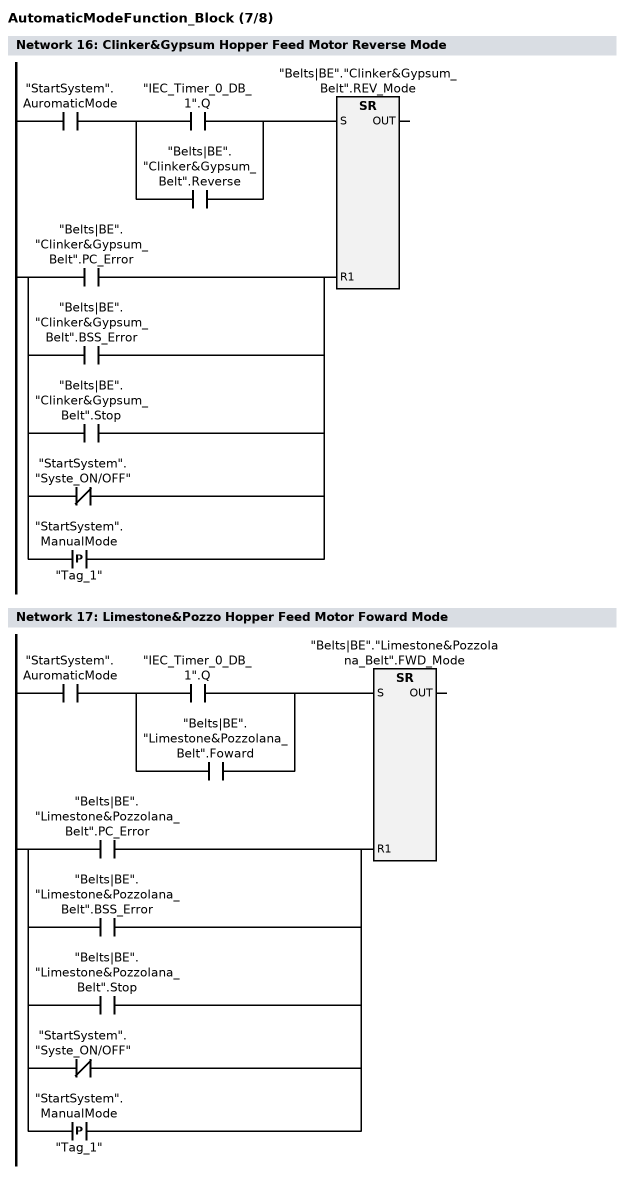
   RUNG wire#powerrail
      Contact( "StartSystem".AuromaticMode )
      wire#w1
      Contact( "IEC_Timer_0_DB_1".Q )
      wire#w2
      S_SR(operand := "Belts|BE"."Clinker&Gypsum_Belt".REV_Mode, r1 := wire#w3)
   END_RUNG
   RUNG wire#w1
      Contact( "Belts|BE"."Clinker&Gypsum_Belt".Reverse )
   END_RUNG wire#w2
   RUNG wire#powerrail
      Contact( "Belts|BE"."Clinker&Gypsum_Belt".PC_Error )
   END_RUNG wire#w3
   RUNG wire#powerrail
      Contact( "Belts|BE"."Clinker&Gypsum_Belt".BSS_Error )
   END_RUNG wire#w3
   RUNG wire#powerrail
      Contact( "Belts|BE"."Clinker&Gypsum_Belt".Stop )
   END_RUNG wire#w3
   RUNG wire#powerrail
      I_Contact( "StartSystem"."Syste_ON/OFF" )
   END_RUNG wire#w3
   RUNG wire#powerrail
      P_Contact(operand := "StartSystem".ManualMode, bit := "Tag_1")
   END_RUNG wire#w3
   // the same network as SCL:
   #_w1 := "StartSystem".ManualMode AND NOT "Tag_1";   // rising edge of "StartSystem".ManualMode
   "Tag_1" := "StartSystem".ManualMode;
   IF "StartSystem".AuromaticMode AND ("IEC_Timer_0_DB_1".Q OR "Belts|BE"."Clinker&Gypsum_Belt".Reverse) THEN
       "Belts|BE"."Clinker&Gypsum_Belt".REV_Mode := TRUE;   // SR flip-flop
   END_IF;
   IF "Belts|BE"."Clinker&Gypsum_Belt".PC_Error OR "Belts|BE"."Clinker&Gypsum_Belt".BSS_Error OR "Belts|BE"."Clinker&Gypsum_Belt".Stop OR NOT "StartSystem"."Syste_ON/OFF" OR #_w1 THEN
       "Belts|BE"."Clinker&Gypsum_Belt".REV_Mode := FALSE;
   END_IF;
END_REGION

REGION Network 17: Limestone&Pozzo Hopper Feed Motor Foward Mode
   RUNG wire#powerrail
      Contact( "StartSystem".AuromaticMode )
      wire#w1
      Contact( "IEC_Timer_0_DB_1".Q )
      wire#w2
      S_SR(operand := "Belts|BE"."Limestone&Pozzolana_Belt".FWD_Mode, r1 := wire#w3)
   END_RUNG
   RUNG wire#w1
      Contact( "Belts|BE"."Limestone&Pozzolana_Belt".Foward )
   END_RUNG wire#w2
   RUNG wire#powerrail
      Contact( "Belts|BE"."Limestone&Pozzolana_Belt".PC_Error )
   END_RUNG wire#w3
   RUNG wire#powerrail
      Contact( "Belts|BE"."Limestone&Pozzolana_Belt".BSS_Error )
   END_RUNG wire#w3
   RUNG wire#powerrail
      Contact( "Belts|BE"."Limestone&Pozzolana_Belt".Stop )
   END_RUNG wire#w3
   RUNG wire#powerrail
      I_Contact( "StartSystem"."Syste_ON/OFF" )
   END_RUNG wire#w3
   RUNG wire#powerrail
      P_Contact(operand := "StartSystem".ManualMode, bit := "Tag_1")
   END_RUNG wire#w3
   // the same network as SCL:
   #_w1 := "StartSystem".ManualMode AND NOT "Tag_1";   // rising edge of "StartSystem".ManualMode
   "Tag_1" := "StartSystem".ManualMode;
   IF "StartSystem".AuromaticMode AND ("IEC_Timer_0_DB_1".Q OR "Belts|BE"."Limestone&Pozzolana_Belt".Foward) THEN
       "Belts|BE"."Limestone&Pozzolana_Belt".FWD_Mode := TRUE;   // SR flip-flop
   END_IF;
   IF "Belts|BE"."Limestone&Pozzolana_Belt".PC_Error OR "Belts|BE"."Limestone&Pozzolana_Belt".BSS_Error OR "Belts|BE"."Limestone&Pozzolana_Belt".Stop OR NOT "StartSystem"."Syste_ON/OFF" OR #_w1 THEN
       "Belts|BE"."Limestone&Pozzolana_Belt".FWD_Mode := FALSE;
   END_IF;
END_REGION

REGION Network 18: Limestone&Pozzo Hopper Feed Motor Reverse Mode
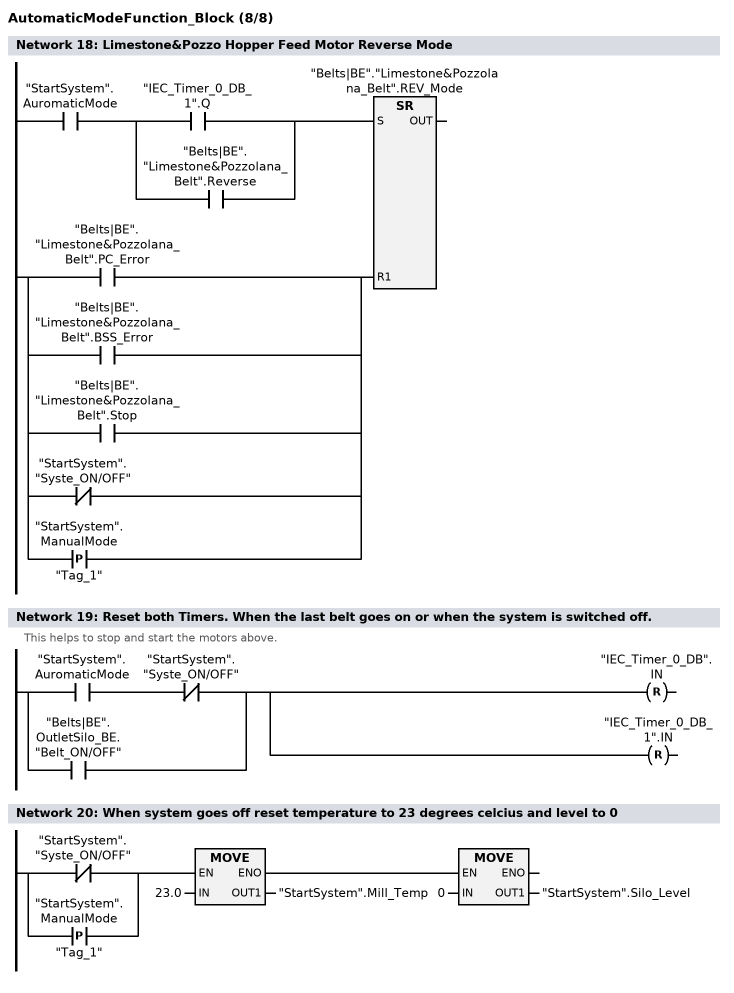
   RUNG wire#powerrail
      Contact( "StartSystem".AuromaticMode )
      wire#w1
      Contact( "IEC_Timer_0_DB_1".Q )
      wire#w2
      S_SR(operand := "Belts|BE"."Limestone&Pozzolana_Belt".REV_Mode, r1 := wire#w3)
   END_RUNG
   RUNG wire#w1
      Contact( "Belts|BE"."Limestone&Pozzolana_Belt".Reverse )
   END_RUNG wire#w2
   RUNG wire#powerrail
      Contact( "Belts|BE"."Limestone&Pozzolana_Belt".PC_Error )
   END_RUNG wire#w3
   RUNG wire#powerrail
      Contact( "Belts|BE"."Limestone&Pozzolana_Belt".BSS_Error )
   END_RUNG wire#w3
   RUNG wire#powerrail
      Contact( "Belts|BE"."Limestone&Pozzolana_Belt".Stop )
   END_RUNG wire#w3
   RUNG wire#powerrail
      I_Contact( "StartSystem"."Syste_ON/OFF" )
   END_RUNG wire#w3
   RUNG wire#powerrail
      P_Contact(operand := "StartSystem".ManualMode, bit := "Tag_1")
   END_RUNG wire#w3
   // the same network as SCL:
   #_w1 := "StartSystem".ManualMode AND NOT "Tag_1";   // rising edge of "StartSystem".ManualMode
   "Tag_1" := "StartSystem".ManualMode;
   IF "StartSystem".AuromaticMode AND ("IEC_Timer_0_DB_1".Q OR "Belts|BE"."Limestone&Pozzolana_Belt".Reverse) THEN
       "Belts|BE"."Limestone&Pozzolana_Belt".REV_Mode := TRUE;   // SR flip-flop
   END_IF;
   IF "Belts|BE"."Limestone&Pozzolana_Belt".PC_Error OR "Belts|BE"."Limestone&Pozzolana_Belt".BSS_Error OR "Belts|BE"."Limestone&Pozzolana_Belt".Stop OR NOT "StartSystem"."Syste_ON/OFF" OR #_w1 THEN
       "Belts|BE"."Limestone&Pozzolana_Belt".REV_Mode := FALSE;
   END_IF;
END_REGION

REGION Network 19: Reset both Timers. When the last belt goes on or when the system is switched off.
   // This helps to stop and start the motors above.
   RUNG wire#powerrail
      Contact( "StartSystem".AuromaticMode )
      I_Contact( "StartSystem"."Syste_ON/OFF" )
      wire#w1
      R_Coil( "IEC_Timer_0_DB".IN )
   END_RUNG
   RUNG wire#powerrail
      Contact( "Belts|BE".OutletSilo_BE."Belt_ON/OFF" )
   END_RUNG wire#w1
   RUNG wire#w1
      R_Coil( "IEC_Timer_0_DB_1".IN )
   END_RUNG
   // the same network as SCL:
   IF ("StartSystem".AuromaticMode AND NOT "StartSystem"."Syste_ON/OFF") OR "Belts|BE".OutletSilo_BE."Belt_ON/OFF" THEN
       "IEC_Timer_0_DB".IN := FALSE;
       "IEC_Timer_0_DB_1".IN := FALSE;
   END_IF;
END_REGION

REGION Network 20: When system goes off reset temperature to 23 degrees celcius and level to 0
   RUNG wire#powerrail
      I_Contact( "StartSystem"."Syste_ON/OFF" )
      wire#w1
      Move(in := 23.0, out1 => "StartSystem".Mill_Temp)
      Move(in := 0, out1 => "StartSystem".Silo_Level)
   END_RUNG
   RUNG wire#powerrail
      P_Contact(operand := "StartSystem".ManualMode, bit := "Tag_1")
   END_RUNG wire#w1
   // the same network as SCL:
   #_w1 := "StartSystem".ManualMode AND NOT "Tag_1";   // rising edge of "StartSystem".ManualMode
   "Tag_1" := "StartSystem".ManualMode;
   IF NOT "StartSystem"."Syste_ON/OFF" OR #_w1 THEN
       "StartSystem".Mill_Temp := 23.0;
       "StartSystem".Silo_Level := 0;
   END_IF;
END_REGION
END_FUNCTION

FUNCTION "Belt_Errors_AutoMode" : Void   // FC7, LAD
{ S7_Optimized_Access := 'TRUE' }
VERSION : 0.1
   VAR_INPUT
      PC : Bool;
      BSS : Bool;
      Reset : Bool;
   END_VAR
   VAR_IN_OUT
      BSS_Error : Bool;
      PC_Error : Bool;
   END_VAR
BEGIN

REGION Network 1: Beltsway error and pull code errors setting and resetting
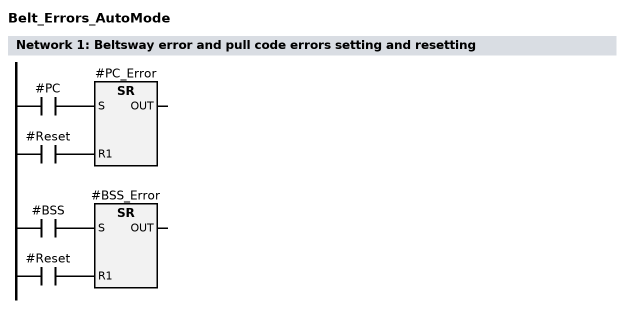
   RUNG wire#powerrail
      Contact( #PC )
      S_SR(operand := #PC_Error, r1 := wire#w1)
   END_RUNG
   RUNG wire#powerrail
      Contact( #Reset )
   END_RUNG wire#w1
   RUNG wire#powerrail
      Contact( #BSS )
      S_SR(operand := #BSS_Error, r1 := wire#w2)
   END_RUNG
   RUNG wire#powerrail
      Contact( #Reset )
   END_RUNG wire#w2
   // the same network as SCL:
   IF #PC THEN
       #PC_Error := TRUE;   // SR flip-flop
   END_IF;
   IF #Reset THEN #PC_Error := FALSE; END_IF;
   IF #BSS THEN
       #BSS_Error := TRUE;   // SR flip-flop
   END_IF;
   IF #Reset THEN #BSS_Error := FALSE; END_IF;
END_REGION
END_FUNCTION

FUNCTION "ErrorHandlingAuto" : Void   // FC8, LAD
{ S7_Optimized_Access := 'TRUE' }
VERSION : 0.1
BEGIN

REGION Network 1: Pozzolana Belt
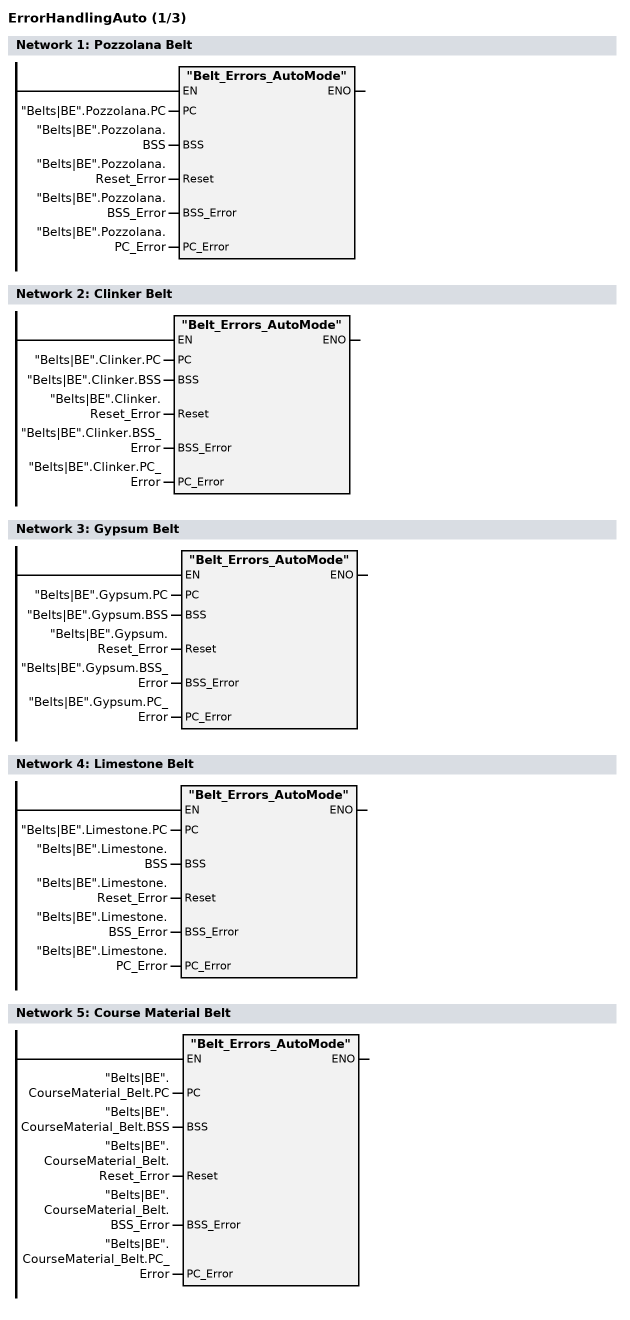
   RUNG wire#powerrail
      "Belt_Errors_AutoMode"(PC := "Belts|BE".Pozzolana.PC, BSS := "Belts|BE".Pozzolana.BSS, Reset := "Belts|BE".Pozzolana.Reset_Error, BSS_Error := "Belts|BE".Pozzolana.BSS_Error, PC_Error := "Belts|BE".Pozzolana.PC_Error)
   END_RUNG
   // the same network as SCL:
   "Belt_Errors_AutoMode"(PC := "Belts|BE".Pozzolana.PC,
                          BSS := "Belts|BE".Pozzolana.BSS,
                          Reset := "Belts|BE".Pozzolana.Reset_Error,
                          BSS_Error := "Belts|BE".Pozzolana.BSS_Error,
                          PC_Error := "Belts|BE".Pozzolana.PC_Error);
END_REGION

REGION Network 2: Clinker Belt
   RUNG wire#powerrail
      "Belt_Errors_AutoMode"(PC := "Belts|BE".Clinker.PC, BSS := "Belts|BE".Clinker.BSS, Reset := "Belts|BE".Clinker.Reset_Error, BSS_Error := "Belts|BE".Clinker.BSS_Error, PC_Error := "Belts|BE".Clinker.PC_Error)
   END_RUNG
   // the same network as SCL:
   "Belt_Errors_AutoMode"(PC := "Belts|BE".Clinker.PC,
                          BSS := "Belts|BE".Clinker.BSS,
                          Reset := "Belts|BE".Clinker.Reset_Error,
                          BSS_Error := "Belts|BE".Clinker.BSS_Error,
                          PC_Error := "Belts|BE".Clinker.PC_Error);
END_REGION

REGION Network 3: Gypsum Belt
   RUNG wire#powerrail
      "Belt_Errors_AutoMode"(PC := "Belts|BE".Gypsum.PC, BSS := "Belts|BE".Gypsum.BSS, Reset := "Belts|BE".Gypsum.Reset_Error, BSS_Error := "Belts|BE".Gypsum.BSS_Error, PC_Error := "Belts|BE".Gypsum.PC_Error)
   END_RUNG
   // the same network as SCL:
   "Belt_Errors_AutoMode"(PC := "Belts|BE".Gypsum.PC,
                          BSS := "Belts|BE".Gypsum.BSS,
                          Reset := "Belts|BE".Gypsum.Reset_Error,
                          BSS_Error := "Belts|BE".Gypsum.BSS_Error,
                          PC_Error := "Belts|BE".Gypsum.PC_Error);
END_REGION

REGION Network 4: Limestone Belt
   RUNG wire#powerrail
      "Belt_Errors_AutoMode"(PC := "Belts|BE".Limestone.PC, BSS := "Belts|BE".Limestone.BSS, Reset := "Belts|BE".Limestone.Reset_Error, BSS_Error := "Belts|BE".Limestone.BSS_Error, PC_Error := "Belts|BE".Limestone.PC_Error)
   END_RUNG
   // the same network as SCL:
   "Belt_Errors_AutoMode"(PC := "Belts|BE".Limestone.PC,
                          BSS := "Belts|BE".Limestone.BSS,
                          Reset := "Belts|BE".Limestone.Reset_Error,
                          BSS_Error := "Belts|BE".Limestone.BSS_Error,
                          PC_Error := "Belts|BE".Limestone.PC_Error);
END_REGION

REGION Network 5: Course Material Belt
   RUNG wire#powerrail
      "Belt_Errors_AutoMode"(PC := "Belts|BE".CourseMaterial_Belt.PC, BSS := "Belts|BE".CourseMaterial_Belt.BSS, Reset := "Belts|BE".CourseMaterial_Belt.Reset_Error, BSS_Error := "Belts|BE".CourseMaterial_Belt.BSS_Error, PC_Error := "Belts|BE".CourseMaterial_Belt.PC_Error)
   END_RUNG
   // the same network as SCL:
   "Belt_Errors_AutoMode"(PC := "Belts|BE".CourseMaterial_Belt.PC,
                          BSS := "Belts|BE".CourseMaterial_Belt.BSS,
                          Reset := "Belts|BE".CourseMaterial_Belt.Reset_Error,
                          BSS_Error := "Belts|BE".CourseMaterial_Belt.BSS_Error,
                          PC_Error := "Belts|BE".CourseMaterial_Belt.PC_Error);
END_REGION

REGION Network 6: Material Inlet Belt
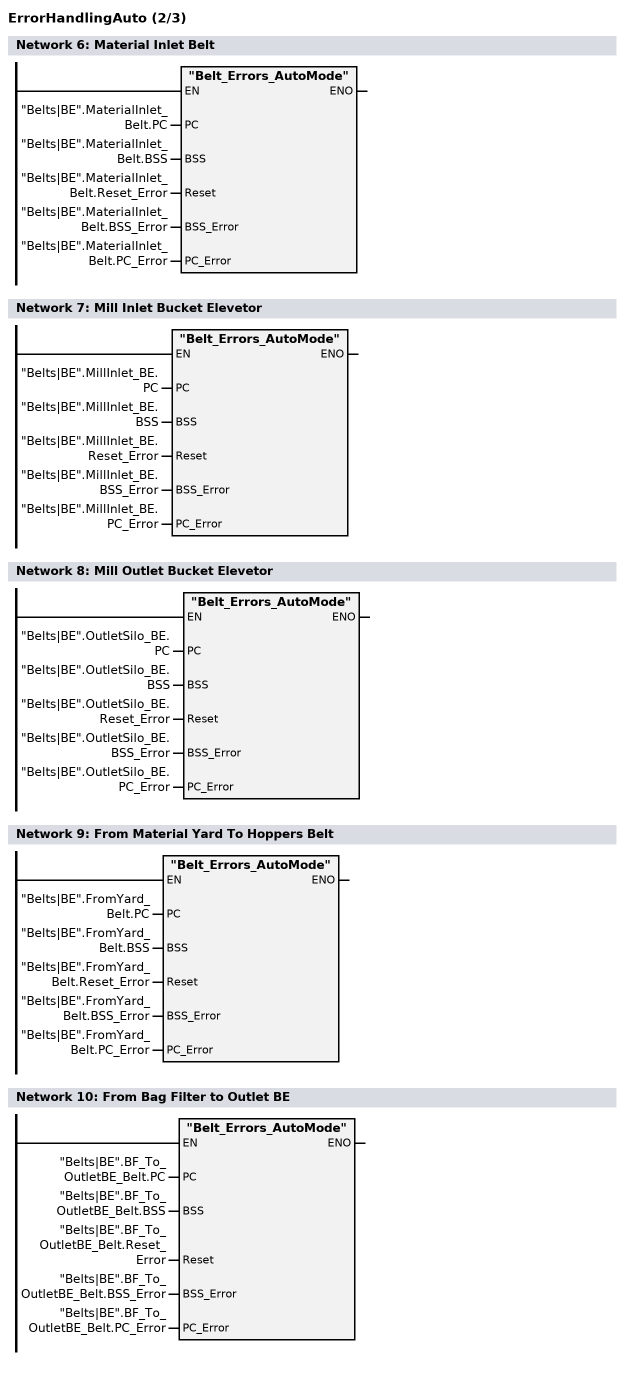
   RUNG wire#powerrail
      "Belt_Errors_AutoMode"(PC := "Belts|BE".MaterialInlet_Belt.PC, BSS := "Belts|BE".MaterialInlet_Belt.BSS, Reset := "Belts|BE".MaterialInlet_Belt.Reset_Error, BSS_Error := "Belts|BE".MaterialInlet_Belt.BSS_Error, PC_Error := "Belts|BE".MaterialInlet_Belt.PC_Error)
   END_RUNG
   // the same network as SCL:
   "Belt_Errors_AutoMode"(PC := "Belts|BE".MaterialInlet_Belt.PC,
                          BSS := "Belts|BE".MaterialInlet_Belt.BSS,
                          Reset := "Belts|BE".MaterialInlet_Belt.Reset_Error,
                          BSS_Error := "Belts|BE".MaterialInlet_Belt.BSS_Error,
                          PC_Error := "Belts|BE".MaterialInlet_Belt.PC_Error);
END_REGION

REGION Network 7: Mill Inlet Bucket Elevetor
   RUNG wire#powerrail
      "Belt_Errors_AutoMode"(PC := "Belts|BE".MillInlet_BE.PC, BSS := "Belts|BE".MillInlet_BE.BSS, Reset := "Belts|BE".MillInlet_BE.Reset_Error, BSS_Error := "Belts|BE".MillInlet_BE.BSS_Error, PC_Error := "Belts|BE".MillInlet_BE.PC_Error)
   END_RUNG
   // the same network as SCL:
   "Belt_Errors_AutoMode"(PC := "Belts|BE".MillInlet_BE.PC,
                          BSS := "Belts|BE".MillInlet_BE.BSS,
                          Reset := "Belts|BE".MillInlet_BE.Reset_Error,
                          BSS_Error := "Belts|BE".MillInlet_BE.BSS_Error,
                          PC_Error := "Belts|BE".MillInlet_BE.PC_Error);
END_REGION

REGION Network 8: Mill Outlet Bucket Elevetor
   RUNG wire#powerrail
      "Belt_Errors_AutoMode"(PC := "Belts|BE".OutletSilo_BE.PC, BSS := "Belts|BE".OutletSilo_BE.BSS, Reset := "Belts|BE".OutletSilo_BE.Reset_Error, BSS_Error := "Belts|BE".OutletSilo_BE.BSS_Error, PC_Error := "Belts|BE".OutletSilo_BE.PC_Error)
   END_RUNG
   // the same network as SCL:
   "Belt_Errors_AutoMode"(PC := "Belts|BE".OutletSilo_BE.PC,
                          BSS := "Belts|BE".OutletSilo_BE.BSS,
                          Reset := "Belts|BE".OutletSilo_BE.Reset_Error,
                          BSS_Error := "Belts|BE".OutletSilo_BE.BSS_Error,
                          PC_Error := "Belts|BE".OutletSilo_BE.PC_Error);
END_REGION

REGION Network 9: From Material Yard To Hoppers Belt
   RUNG wire#powerrail
      "Belt_Errors_AutoMode"(PC := "Belts|BE".FromYard_Belt.PC, BSS := "Belts|BE".FromYard_Belt.BSS, Reset := "Belts|BE".FromYard_Belt.Reset_Error, BSS_Error := "Belts|BE".FromYard_Belt.BSS_Error, PC_Error := "Belts|BE".FromYard_Belt.PC_Error)
   END_RUNG
   // the same network as SCL:
   "Belt_Errors_AutoMode"(PC := "Belts|BE".FromYard_Belt.PC,
                          BSS := "Belts|BE".FromYard_Belt.BSS,
                          Reset := "Belts|BE".FromYard_Belt.Reset_Error,
                          BSS_Error := "Belts|BE".FromYard_Belt.BSS_Error,
                          PC_Error := "Belts|BE".FromYard_Belt.PC_Error);
END_REGION

REGION Network 10: From Bag Filter to Outlet BE
   RUNG wire#powerrail
      "Belt_Errors_AutoMode"(PC := "Belts|BE".BF_To_OutletBE_Belt.PC, BSS := "Belts|BE".BF_To_OutletBE_Belt.BSS, Reset := "Belts|BE".BF_To_OutletBE_Belt.Reset_Error, BSS_Error := "Belts|BE".BF_To_OutletBE_Belt.BSS_Error, PC_Error := "Belts|BE".BF_To_OutletBE_Belt.PC_Error)
   END_RUNG
   // the same network as SCL:
   "Belt_Errors_AutoMode"(PC := "Belts|BE".BF_To_OutletBE_Belt.PC,
                          BSS := "Belts|BE".BF_To_OutletBE_Belt.BSS,
                          Reset := "Belts|BE".BF_To_OutletBE_Belt.Reset_Error,
                          BSS_Error := "Belts|BE".BF_To_OutletBE_Belt.BSS_Error,
                          PC_Error := "Belts|BE".BF_To_OutletBE_Belt.PC_Error);
END_REGION

REGION Network 11: Clinker&Gypsum Belt
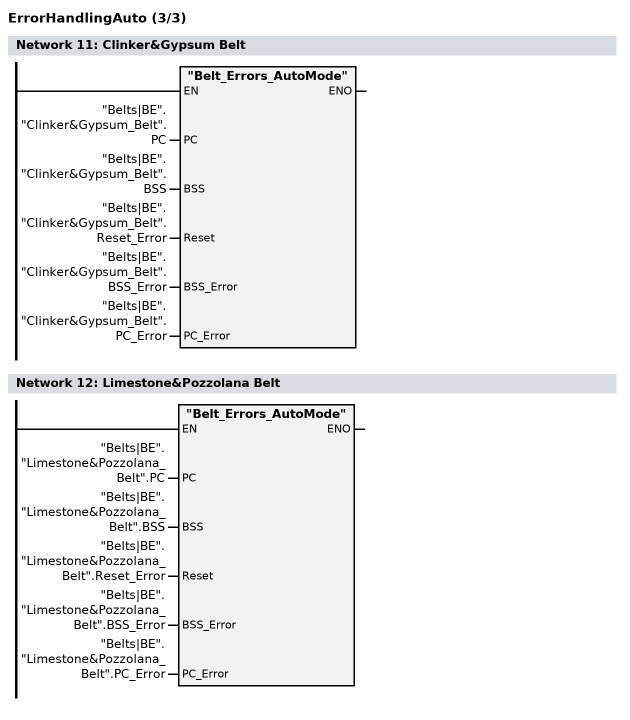
   RUNG wire#powerrail
      "Belt_Errors_AutoMode"(PC := "Belts|BE"."Clinker&Gypsum_Belt".PC, BSS := "Belts|BE"."Clinker&Gypsum_Belt".BSS, Reset := "Belts|BE"."Clinker&Gypsum_Belt".Reset_Error, BSS_Error := "Belts|BE"."Clinker&Gypsum_Belt".BSS_Error, PC_Error := "Belts|BE"."Clinker&Gypsum_Belt".PC_Error)
   END_RUNG
   // the same network as SCL:
   "Belt_Errors_AutoMode"(PC := "Belts|BE"."Clinker&Gypsum_Belt".PC,
                          BSS := "Belts|BE"."Clinker&Gypsum_Belt".BSS,
                          Reset := "Belts|BE"."Clinker&Gypsum_Belt".Reset_Error,
                          BSS_Error := "Belts|BE"."Clinker&Gypsum_Belt".BSS_Error,
                          PC_Error := "Belts|BE"."Clinker&Gypsum_Belt".PC_Error);
END_REGION

REGION Network 12: Limestone&Pozzolana Belt
   RUNG wire#powerrail
      "Belt_Errors_AutoMode"(PC := "Belts|BE"."Limestone&Pozzolana_Belt".PC, BSS := "Belts|BE"."Limestone&Pozzolana_Belt".BSS, Reset := "Belts|BE"."Limestone&Pozzolana_Belt".Reset_Error, BSS_Error := "Belts|BE"."Limestone&Pozzolana_Belt".BSS_Error, PC_Error := "Belts|BE"."Limestone&Pozzolana_Belt".PC_Error)
   END_RUNG
   // the same network as SCL:
   "Belt_Errors_AutoMode"(PC := "Belts|BE"."Limestone&Pozzolana_Belt".PC,
                          BSS := "Belts|BE"."Limestone&Pozzolana_Belt".BSS,
                          Reset := "Belts|BE"."Limestone&Pozzolana_Belt".Reset_Error,
                          BSS_Error := "Belts|BE"."Limestone&Pozzolana_Belt".BSS_Error,
                          PC_Error := "Belts|BE"."Limestone&Pozzolana_Belt".PC_Error);
END_REGION
END_FUNCTION

// folder: Manual_Mode

FUNCTION "ManualModeFunction_Block" : Void   // FC1, LAD
{ S7_Optimized_Access := 'TRUE' }
VERSION : 0.1
BEGIN

REGION Network 1: Starting the main bag filter
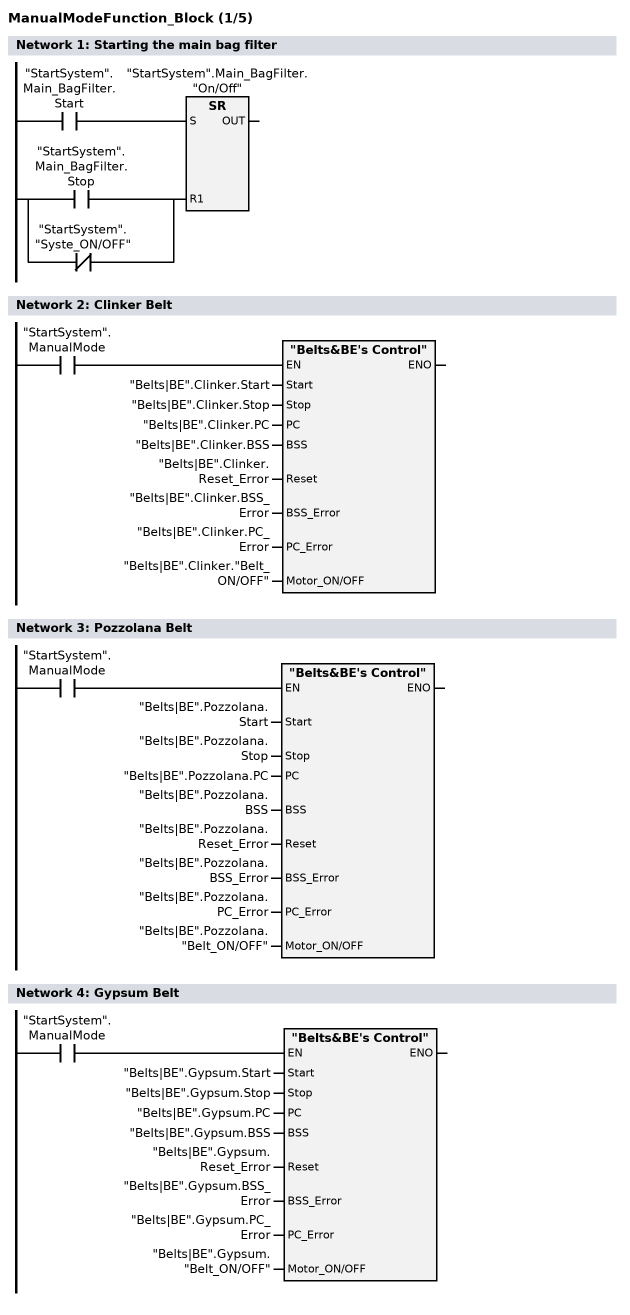
   RUNG wire#powerrail
      Contact( "StartSystem".Main_BagFilter.Start )
      S_SR(operand := "StartSystem".Main_BagFilter."On/Off", r1 := wire#w1)
   END_RUNG
   RUNG wire#powerrail
      Contact( "StartSystem".Main_BagFilter.Stop )
   END_RUNG wire#w1
   RUNG wire#powerrail
      I_Contact( "StartSystem"."Syste_ON/OFF" )
   END_RUNG wire#w1
   // the same network as SCL:
   IF "StartSystem".Main_BagFilter.Start THEN
       "StartSystem".Main_BagFilter."On/Off" := TRUE;   // SR flip-flop
   END_IF;
   IF "StartSystem".Main_BagFilter.Stop OR NOT "StartSystem"."Syste_ON/OFF" THEN
       "StartSystem".Main_BagFilter."On/Off" := FALSE;
   END_IF;
END_REGION

REGION Network 2: Clinker Belt
   RUNG wire#powerrail
      Contact( "StartSystem".ManualMode )
      "Belts&BE's Control"(Start := "Belts|BE".Clinker.Start, Stop := "Belts|BE".Clinker.Stop, PC := "Belts|BE".Clinker.PC, BSS := "Belts|BE".Clinker.BSS, Reset := "Belts|BE".Clinker.Reset_Error, BSS_Error := "Belts|BE".Clinker.BSS_Error, PC_Error := "Belts|BE".Clinker.PC_Error, "Motor_ON/OFF" := "Belts|BE".Clinker."Belt_ON/OFF")
   END_RUNG
   // the same network as SCL:
   IF "StartSystem".ManualMode THEN
       "Belts&BE's Control"(Start := "Belts|BE".Clinker.Start,
                            Stop := "Belts|BE".Clinker.Stop,
                            PC := "Belts|BE".Clinker.PC,
                            BSS := "Belts|BE".Clinker.BSS,
                            Reset := "Belts|BE".Clinker.Reset_Error,
                            BSS_Error := "Belts|BE".Clinker.BSS_Error,
                            PC_Error := "Belts|BE".Clinker.PC_Error,
                            "Motor_ON/OFF" := "Belts|BE".Clinker."Belt_ON/OFF");
   END_IF;
END_REGION

REGION Network 3: Pozzolana Belt
   RUNG wire#powerrail
      Contact( "StartSystem".ManualMode )
      "Belts&BE's Control"(Start := "Belts|BE".Pozzolana.Start, Stop := "Belts|BE".Pozzolana.Stop, PC := "Belts|BE".Pozzolana.PC, BSS := "Belts|BE".Pozzolana.BSS, Reset := "Belts|BE".Pozzolana.Reset_Error, BSS_Error := "Belts|BE".Pozzolana.BSS_Error, PC_Error := "Belts|BE".Pozzolana.PC_Error, "Motor_ON/OFF" := "Belts|BE".Pozzolana."Belt_ON/OFF")
   END_RUNG
   // the same network as SCL:
   IF "StartSystem".ManualMode THEN
       "Belts&BE's Control"(Start := "Belts|BE".Pozzolana.Start,
                            Stop := "Belts|BE".Pozzolana.Stop,
                            PC := "Belts|BE".Pozzolana.PC,
                            BSS := "Belts|BE".Pozzolana.BSS,
                            Reset := "Belts|BE".Pozzolana.Reset_Error,
                            BSS_Error := "Belts|BE".Pozzolana.BSS_Error,
                            PC_Error := "Belts|BE".Pozzolana.PC_Error,
                            "Motor_ON/OFF" := "Belts|BE".Pozzolana."Belt_ON/OFF");
   END_IF;
END_REGION

REGION Network 4: Gypsum Belt
   RUNG wire#powerrail
      Contact( "StartSystem".ManualMode )
      "Belts&BE's Control"(Start := "Belts|BE".Gypsum.Start, Stop := "Belts|BE".Gypsum.Stop, PC := "Belts|BE".Gypsum.PC, BSS := "Belts|BE".Gypsum.BSS, Reset := "Belts|BE".Gypsum.Reset_Error, BSS_Error := "Belts|BE".Gypsum.BSS_Error, PC_Error := "Belts|BE".Gypsum.PC_Error, "Motor_ON/OFF" := "Belts|BE".Gypsum."Belt_ON/OFF")
   END_RUNG
   // the same network as SCL:
   IF "StartSystem".ManualMode THEN
       "Belts&BE's Control"(Start := "Belts|BE".Gypsum.Start,
                            Stop := "Belts|BE".Gypsum.Stop,
                            PC := "Belts|BE".Gypsum.PC,
                            BSS := "Belts|BE".Gypsum.BSS,
                            Reset := "Belts|BE".Gypsum.Reset_Error,
                            BSS_Error := "Belts|BE".Gypsum.BSS_Error,
                            PC_Error := "Belts|BE".Gypsum.PC_Error,
                            "Motor_ON/OFF" := "Belts|BE".Gypsum."Belt_ON/OFF");
   END_IF;
END_REGION

REGION Network 5: Limestone
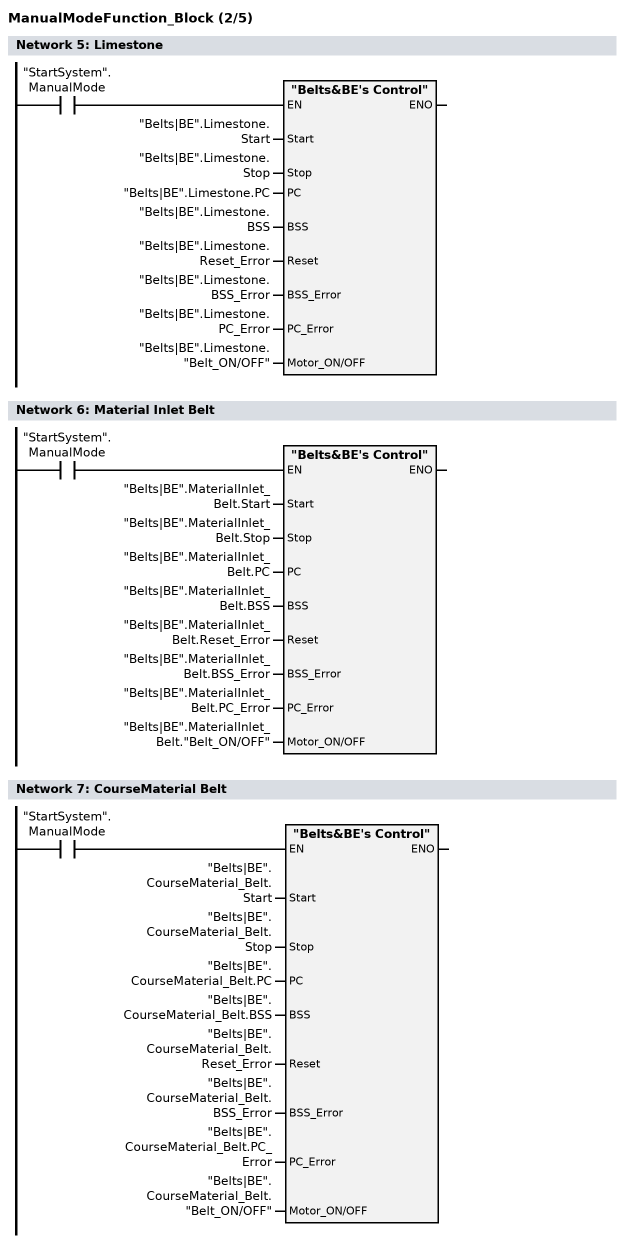
   RUNG wire#powerrail
      Contact( "StartSystem".ManualMode )
      "Belts&BE's Control"(Start := "Belts|BE".Limestone.Start, Stop := "Belts|BE".Limestone.Stop, PC := "Belts|BE".Limestone.PC, BSS := "Belts|BE".Limestone.BSS, Reset := "Belts|BE".Limestone.Reset_Error, BSS_Error := "Belts|BE".Limestone.BSS_Error, PC_Error := "Belts|BE".Limestone.PC_Error, "Motor_ON/OFF" := "Belts|BE".Limestone."Belt_ON/OFF")
   END_RUNG
   // the same network as SCL:
   IF "StartSystem".ManualMode THEN
       "Belts&BE's Control"(Start := "Belts|BE".Limestone.Start,
                            Stop := "Belts|BE".Limestone.Stop,
                            PC := "Belts|BE".Limestone.PC,
                            BSS := "Belts|BE".Limestone.BSS,
                            Reset := "Belts|BE".Limestone.Reset_Error,
                            BSS_Error := "Belts|BE".Limestone.BSS_Error,
                            PC_Error := "Belts|BE".Limestone.PC_Error,
                            "Motor_ON/OFF" := "Belts|BE".Limestone."Belt_ON/OFF");
   END_IF;
END_REGION

REGION Network 6: Material Inlet Belt
   RUNG wire#powerrail
      Contact( "StartSystem".ManualMode )
      "Belts&BE's Control"(Start := "Belts|BE".MaterialInlet_Belt.Start, Stop := "Belts|BE".MaterialInlet_Belt.Stop, PC := "Belts|BE".MaterialInlet_Belt.PC, BSS := "Belts|BE".MaterialInlet_Belt.BSS, Reset := "Belts|BE".MaterialInlet_Belt.Reset_Error, BSS_Error := "Belts|BE".MaterialInlet_Belt.BSS_Error, PC_Error := "Belts|BE".MaterialInlet_Belt.PC_Error, "Motor_ON/OFF" := "Belts|BE".MaterialInlet_Belt."Belt_ON/OFF")
   END_RUNG
   // the same network as SCL:
   IF "StartSystem".ManualMode THEN
       "Belts&BE's Control"(Start := "Belts|BE".MaterialInlet_Belt.Start,
                            Stop := "Belts|BE".MaterialInlet_Belt.Stop,
                            PC := "Belts|BE".MaterialInlet_Belt.PC,
                            BSS := "Belts|BE".MaterialInlet_Belt.BSS,
                            Reset := "Belts|BE".MaterialInlet_Belt.Reset_Error,
                            BSS_Error := "Belts|BE".MaterialInlet_Belt.BSS_Error,
                            PC_Error := "Belts|BE".MaterialInlet_Belt.PC_Error,
                            "Motor_ON/OFF" := "Belts|BE".MaterialInlet_Belt."Belt_ON/OFF");
   END_IF;
END_REGION

REGION Network 7: CourseMaterial Belt
   RUNG wire#powerrail
      Contact( "StartSystem".ManualMode )
      "Belts&BE's Control"(Start := "Belts|BE".CourseMaterial_Belt.Start, Stop := "Belts|BE".CourseMaterial_Belt.Stop, PC := "Belts|BE".CourseMaterial_Belt.PC, BSS := "Belts|BE".CourseMaterial_Belt.BSS, Reset := "Belts|BE".CourseMaterial_Belt.Reset_Error, BSS_Error := "Belts|BE".CourseMaterial_Belt.BSS_Error, PC_Error := "Belts|BE".CourseMaterial_Belt.PC_Error, "Motor_ON/OFF" := "Belts|BE".CourseMaterial_Belt."Belt_ON/OFF")
   END_RUNG
   // the same network as SCL:
   IF "StartSystem".ManualMode THEN
       "Belts&BE's Control"(Start := "Belts|BE".CourseMaterial_Belt.Start,
                            Stop := "Belts|BE".CourseMaterial_Belt.Stop,
                            PC := "Belts|BE".CourseMaterial_Belt.PC,
                            BSS := "Belts|BE".CourseMaterial_Belt.BSS,
                            Reset := "Belts|BE".CourseMaterial_Belt.Reset_Error,
                            BSS_Error := "Belts|BE".CourseMaterial_Belt.BSS_Error,
                            PC_Error := "Belts|BE".CourseMaterial_Belt.PC_Error,
                            "Motor_ON/OFF" := "Belts|BE".CourseMaterial_Belt."Belt_ON/OFF");
   END_IF;
END_REGION

REGION Network 8: Mill Inlet Belt
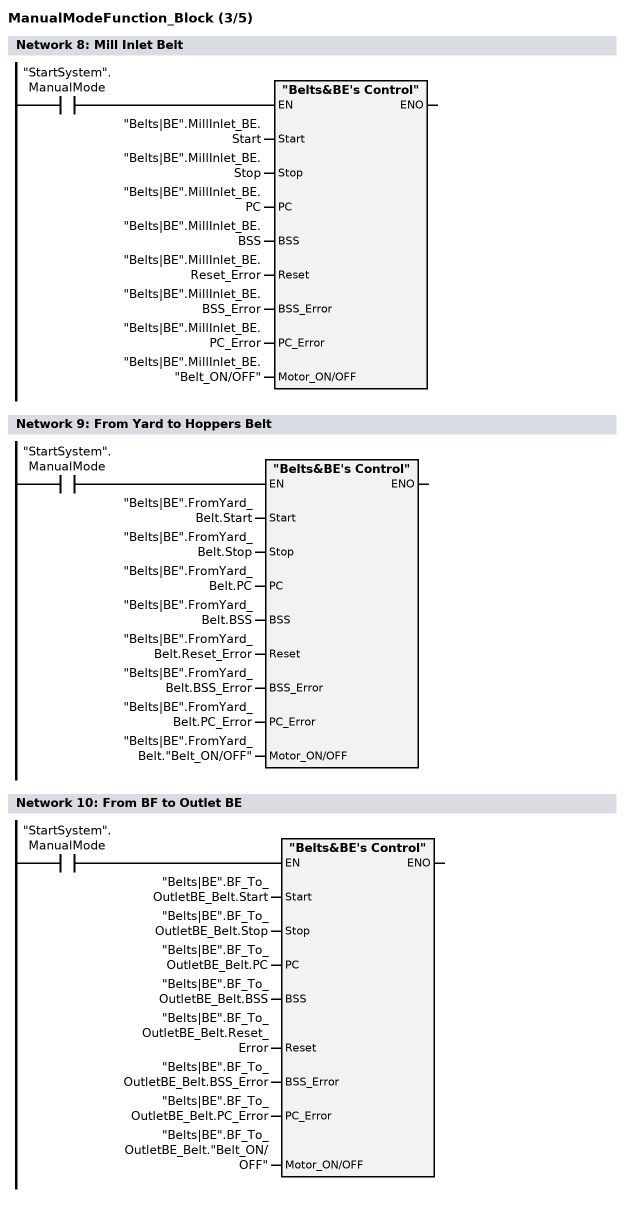
   RUNG wire#powerrail
      Contact( "StartSystem".ManualMode )
      "Belts&BE's Control"(Start := "Belts|BE".MillInlet_BE.Start, Stop := "Belts|BE".MillInlet_BE.Stop, PC := "Belts|BE".MillInlet_BE.PC, BSS := "Belts|BE".MillInlet_BE.BSS, Reset := "Belts|BE".MillInlet_BE.Reset_Error, BSS_Error := "Belts|BE".MillInlet_BE.BSS_Error, PC_Error := "Belts|BE".MillInlet_BE.PC_Error, "Motor_ON/OFF" := "Belts|BE".MillInlet_BE."Belt_ON/OFF")
   END_RUNG
   // the same network as SCL:
   IF "StartSystem".ManualMode THEN
       "Belts&BE's Control"(Start := "Belts|BE".MillInlet_BE.Start,
                            Stop := "Belts|BE".MillInlet_BE.Stop,
                            PC := "Belts|BE".MillInlet_BE.PC,
                            BSS := "Belts|BE".MillInlet_BE.BSS,
                            Reset := "Belts|BE".MillInlet_BE.Reset_Error,
                            BSS_Error := "Belts|BE".MillInlet_BE.BSS_Error,
                            PC_Error := "Belts|BE".MillInlet_BE.PC_Error,
                            "Motor_ON/OFF" := "Belts|BE".MillInlet_BE."Belt_ON/OFF");
   END_IF;
END_REGION

REGION Network 9: From Yard to Hoppers Belt
   RUNG wire#powerrail
      Contact( "StartSystem".ManualMode )
      "Belts&BE's Control"(Start := "Belts|BE".FromYard_Belt.Start, Stop := "Belts|BE".FromYard_Belt.Stop, PC := "Belts|BE".FromYard_Belt.PC, BSS := "Belts|BE".FromYard_Belt.BSS, Reset := "Belts|BE".FromYard_Belt.Reset_Error, BSS_Error := "Belts|BE".FromYard_Belt.BSS_Error, PC_Error := "Belts|BE".FromYard_Belt.PC_Error, "Motor_ON/OFF" := "Belts|BE".FromYard_Belt."Belt_ON/OFF")
   END_RUNG
   // the same network as SCL:
   IF "StartSystem".ManualMode THEN
       "Belts&BE's Control"(Start := "Belts|BE".FromYard_Belt.Start,
                            Stop := "Belts|BE".FromYard_Belt.Stop,
                            PC := "Belts|BE".FromYard_Belt.PC,
                            BSS := "Belts|BE".FromYard_Belt.BSS,
                            Reset := "Belts|BE".FromYard_Belt.Reset_Error,
                            BSS_Error := "Belts|BE".FromYard_Belt.BSS_Error,
                            PC_Error := "Belts|BE".FromYard_Belt.PC_Error,
                            "Motor_ON/OFF" := "Belts|BE".FromYard_Belt."Belt_ON/OFF");
   END_IF;
END_REGION

REGION Network 10: From BF to Outlet BE
   RUNG wire#powerrail
      Contact( "StartSystem".ManualMode )
      "Belts&BE's Control"(Start := "Belts|BE".BF_To_OutletBE_Belt.Start, Stop := "Belts|BE".BF_To_OutletBE_Belt.Stop, PC := "Belts|BE".BF_To_OutletBE_Belt.PC, BSS := "Belts|BE".BF_To_OutletBE_Belt.BSS, Reset := "Belts|BE".BF_To_OutletBE_Belt.Reset_Error, BSS_Error := "Belts|BE".BF_To_OutletBE_Belt.BSS_Error, PC_Error := "Belts|BE".BF_To_OutletBE_Belt.PC_Error, "Motor_ON/OFF" := "Belts|BE".BF_To_OutletBE_Belt."Belt_ON/OFF")
   END_RUNG
   // the same network as SCL:
   IF "StartSystem".ManualMode THEN
       "Belts&BE's Control"(Start := "Belts|BE".BF_To_OutletBE_Belt.Start,
                            Stop := "Belts|BE".BF_To_OutletBE_Belt.Stop,
                            PC := "Belts|BE".BF_To_OutletBE_Belt.PC,
                            BSS := "Belts|BE".BF_To_OutletBE_Belt.BSS,
                            Reset := "Belts|BE".BF_To_OutletBE_Belt.Reset_Error,
                            BSS_Error := "Belts|BE".BF_To_OutletBE_Belt.BSS_Error,
                            PC_Error := "Belts|BE".BF_To_OutletBE_Belt.PC_Error,
                            "Motor_ON/OFF" := "Belts|BE".BF_To_OutletBE_Belt."Belt_ON/OFF");
   END_IF;
END_REGION

REGION Network 11: Clinker&Gypsum FWD/REV
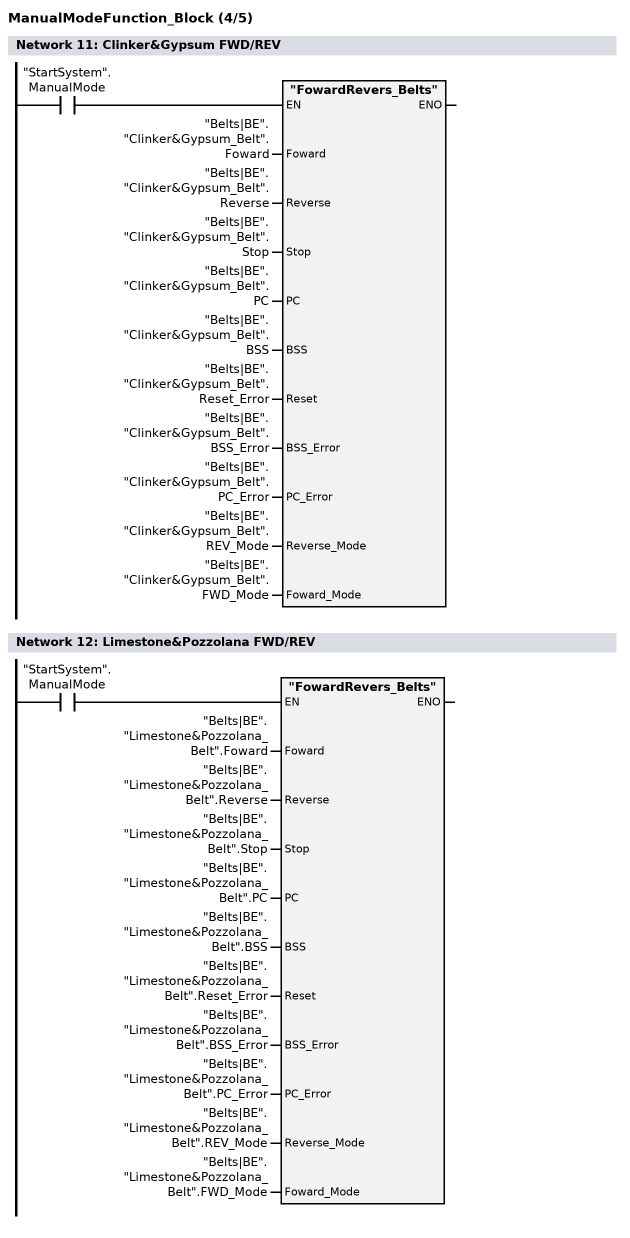
   RUNG wire#powerrail
      Contact( "StartSystem".ManualMode )
      "FowardRevers_Belts"(Foward := "Belts|BE"."Clinker&Gypsum_Belt".Foward, Reverse := "Belts|BE"."Clinker&Gypsum_Belt".Reverse, Stop := "Belts|BE"."Clinker&Gypsum_Belt".Stop, PC := "Belts|BE"."Clinker&Gypsum_Belt".PC, BSS := "Belts|BE"."Clinker&Gypsum_Belt".BSS, Reset := "Belts|BE"."Clinker&Gypsum_Belt".Reset_Error, BSS_Error := "Belts|BE"."Clinker&Gypsum_Belt".BSS_Error, PC_Error := "Belts|BE"."Clinker&Gypsum_Belt".PC_Error, Reverse_Mode := "Belts|BE"."Clinker&Gypsum_Belt".REV_Mode, Foward_Mode := "Belts|BE"."Clinker&Gypsum_Belt".FWD_Mode)
   END_RUNG
   // the same network as SCL:
   IF "StartSystem".ManualMode THEN
       "FowardRevers_Belts"(Foward := "Belts|BE"."Clinker&Gypsum_Belt".Foward,
                            Reverse := "Belts|BE"."Clinker&Gypsum_Belt".Reverse,
                            Stop := "Belts|BE"."Clinker&Gypsum_Belt".Stop,
                            PC := "Belts|BE"."Clinker&Gypsum_Belt".PC,
                            BSS := "Belts|BE"."Clinker&Gypsum_Belt".BSS,
                            Reset := "Belts|BE"."Clinker&Gypsum_Belt".Reset_Error,
                            BSS_Error := "Belts|BE"."Clinker&Gypsum_Belt".BSS_Error,
                            PC_Error := "Belts|BE"."Clinker&Gypsum_Belt".PC_Error,
                            Reverse_Mode := "Belts|BE"."Clinker&Gypsum_Belt".REV_Mode,
                            Foward_Mode := "Belts|BE"."Clinker&Gypsum_Belt".FWD_Mode);
   END_IF;
END_REGION

REGION Network 12: Limestone&Pozzolana FWD/REV
   RUNG wire#powerrail
      Contact( "StartSystem".ManualMode )
      "FowardRevers_Belts"(Foward := "Belts|BE"."Limestone&Pozzolana_Belt".Foward, Reverse := "Belts|BE"."Limestone&Pozzolana_Belt".Reverse, Stop := "Belts|BE"."Limestone&Pozzolana_Belt".Stop, PC := "Belts|BE"."Limestone&Pozzolana_Belt".PC, BSS := "Belts|BE"."Limestone&Pozzolana_Belt".BSS, Reset := "Belts|BE"."Limestone&Pozzolana_Belt".Reset_Error, BSS_Error := "Belts|BE"."Limestone&Pozzolana_Belt".BSS_Error, PC_Error := "Belts|BE"."Limestone&Pozzolana_Belt".PC_Error, Reverse_Mode := "Belts|BE"."Limestone&Pozzolana_Belt".REV_Mode, Foward_Mode := "Belts|BE"."Limestone&Pozzolana_Belt".FWD_Mode)
   END_RUNG
   // the same network as SCL:
   IF "StartSystem".ManualMode THEN
       "FowardRevers_Belts"(Foward := "Belts|BE"."Limestone&Pozzolana_Belt".Foward,
                            Reverse := "Belts|BE"."Limestone&Pozzolana_Belt".Reverse,
                            Stop := "Belts|BE"."Limestone&Pozzolana_Belt".Stop,
                            PC := "Belts|BE"."Limestone&Pozzolana_Belt".PC,
                            BSS := "Belts|BE"."Limestone&Pozzolana_Belt".BSS,
                            Reset := "Belts|BE"."Limestone&Pozzolana_Belt".Reset_Error,
                            BSS_Error := "Belts|BE"."Limestone&Pozzolana_Belt".BSS_Error,
                            PC_Error := "Belts|BE"."Limestone&Pozzolana_Belt".PC_Error,
                            Reverse_Mode := "Belts|BE"."Limestone&Pozzolana_Belt".REV_Mode,
                            Foward_Mode := "Belts|BE"."Limestone&Pozzolana_Belt".FWD_Mode);
   END_IF;
END_REGION

REGION Network 13: Outlet to Silo BE
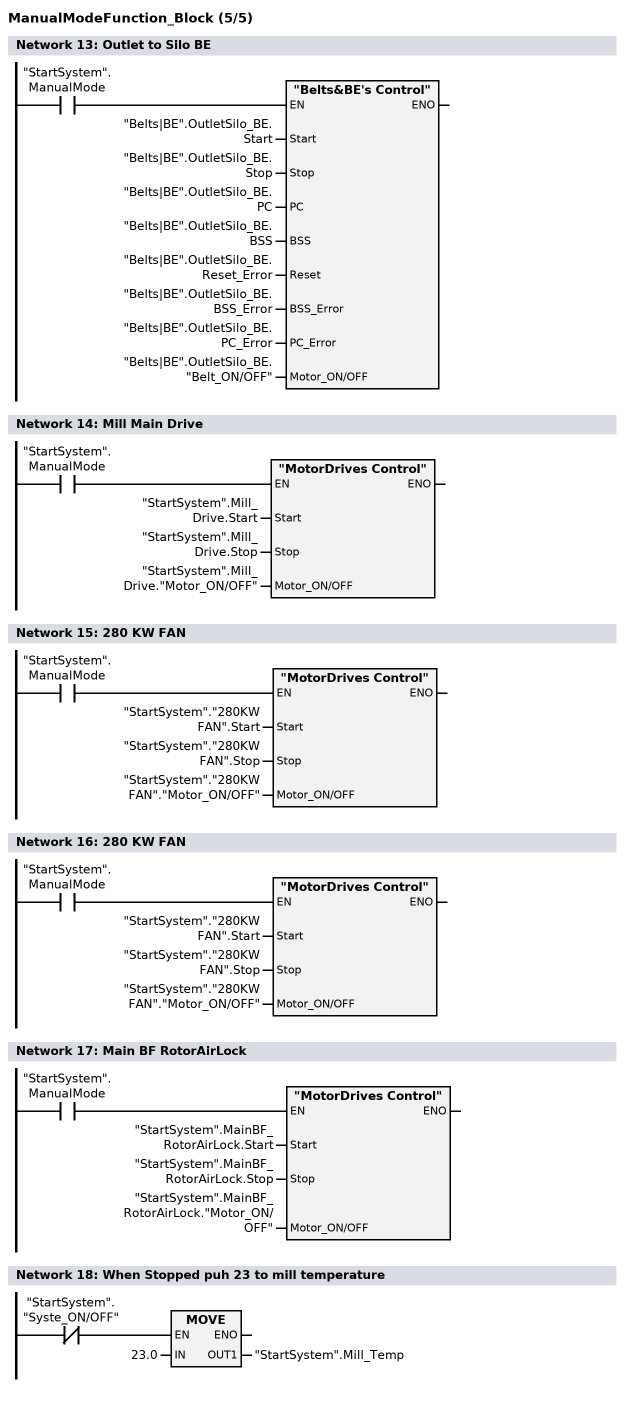
   RUNG wire#powerrail
      Contact( "StartSystem".ManualMode )
      "Belts&BE's Control"(Start := "Belts|BE".OutletSilo_BE.Start, Stop := "Belts|BE".OutletSilo_BE.Stop, PC := "Belts|BE".OutletSilo_BE.PC, BSS := "Belts|BE".OutletSilo_BE.BSS, Reset := "Belts|BE".OutletSilo_BE.Reset_Error, BSS_Error := "Belts|BE".OutletSilo_BE.BSS_Error, PC_Error := "Belts|BE".OutletSilo_BE.PC_Error, "Motor_ON/OFF" := "Belts|BE".OutletSilo_BE."Belt_ON/OFF")
   END_RUNG
   // the same network as SCL:
   IF "StartSystem".ManualMode THEN
       "Belts&BE's Control"(Start := "Belts|BE".OutletSilo_BE.Start,
                            Stop := "Belts|BE".OutletSilo_BE.Stop,
                            PC := "Belts|BE".OutletSilo_BE.PC,
                            BSS := "Belts|BE".OutletSilo_BE.BSS,
                            Reset := "Belts|BE".OutletSilo_BE.Reset_Error,
                            BSS_Error := "Belts|BE".OutletSilo_BE.BSS_Error,
                            PC_Error := "Belts|BE".OutletSilo_BE.PC_Error,
                            "Motor_ON/OFF" := "Belts|BE".OutletSilo_BE."Belt_ON/OFF");
   END_IF;
END_REGION

REGION Network 14: Mill Main Drive
   RUNG wire#powerrail
      Contact( "StartSystem".ManualMode )
      "MotorDrives Control"(Start := "StartSystem".Mill_Drive.Start, Stop := "StartSystem".Mill_Drive.Stop, "Motor_ON/OFF" := "StartSystem".Mill_Drive."Motor_ON/OFF")
   END_RUNG
   // the same network as SCL:
   IF "StartSystem".ManualMode THEN
       "MotorDrives Control"(Start := "StartSystem".Mill_Drive.Start,
                             Stop := "StartSystem".Mill_Drive.Stop,
                             "Motor_ON/OFF" := "StartSystem".Mill_Drive."Motor_ON/OFF");
   END_IF;
END_REGION

REGION Network 15: 280 KW FAN
   RUNG wire#powerrail
      Contact( "StartSystem".ManualMode )
      "MotorDrives Control"(Start := "StartSystem"."280KW FAN".Start, Stop := "StartSystem"."280KW FAN".Stop, "Motor_ON/OFF" := "StartSystem"."280KW FAN"."Motor_ON/OFF")
   END_RUNG
   // the same network as SCL:
   IF "StartSystem".ManualMode THEN
       "MotorDrives Control"(Start := "StartSystem"."280KW FAN".Start,
                             Stop := "StartSystem"."280KW FAN".Stop,
                             "Motor_ON/OFF" := "StartSystem"."280KW FAN"."Motor_ON/OFF");
   END_IF;
END_REGION

REGION Network 16: 280 KW FAN
   RUNG wire#powerrail
      Contact( "StartSystem".ManualMode )
      "MotorDrives Control"(Start := "StartSystem"."280KW FAN".Start, Stop := "StartSystem"."280KW FAN".Stop, "Motor_ON/OFF" := "StartSystem"."280KW FAN"."Motor_ON/OFF")
   END_RUNG
   // the same network as SCL:
   IF "StartSystem".ManualMode THEN
       "MotorDrives Control"(Start := "StartSystem"."280KW FAN".Start,
                             Stop := "StartSystem"."280KW FAN".Stop,
                             "Motor_ON/OFF" := "StartSystem"."280KW FAN"."Motor_ON/OFF");
   END_IF;
END_REGION

REGION Network 17: Main BF RotorAirLock
   RUNG wire#powerrail
      Contact( "StartSystem".ManualMode )
      "MotorDrives Control"(Start := "StartSystem".MainBF_RotorAirLock.Start, Stop := "StartSystem".MainBF_RotorAirLock.Stop, "Motor_ON/OFF" := "StartSystem".MainBF_RotorAirLock."Motor_ON/OFF")
   END_RUNG
   // the same network as SCL:
   IF "StartSystem".ManualMode THEN
       "MotorDrives Control"(Start := "StartSystem".MainBF_RotorAirLock.Start,
                             Stop := "StartSystem".MainBF_RotorAirLock.Stop,
                             "Motor_ON/OFF" := "StartSystem".MainBF_RotorAirLock."Motor_ON/OFF");
   END_IF;
END_REGION

REGION Network 18: When Stopped puh 23 to mill temperature
   RUNG wire#powerrail
      I_Contact( "StartSystem"."Syste_ON/OFF" )
      Move(in := 23.0, out1 => "StartSystem".Mill_Temp)
   END_RUNG
   // the same network as SCL:
   IF NOT "StartSystem"."Syste_ON/OFF" THEN "StartSystem".Mill_Temp := 23.0; END_IF;
END_REGION
END_FUNCTION

FUNCTION "Belts&BE's Control" : Void   // FC3, LAD
{ S7_Optimized_Access := 'TRUE' }
VERSION : 0.1
   VAR_INPUT
      Start : Bool;
      Stop : Bool;
      PC : Bool;
      BSS : Bool;
      Reset : Bool;
   END_VAR
   VAR_IN_OUT
      BSS_Error : Bool;
      PC_Error : Bool;
      "Motor_ON/OFF" : Bool;
   END_VAR
   VAR_TEMP
      Hold_On : Bool;
   END_VAR
BEGIN

REGION Network 1
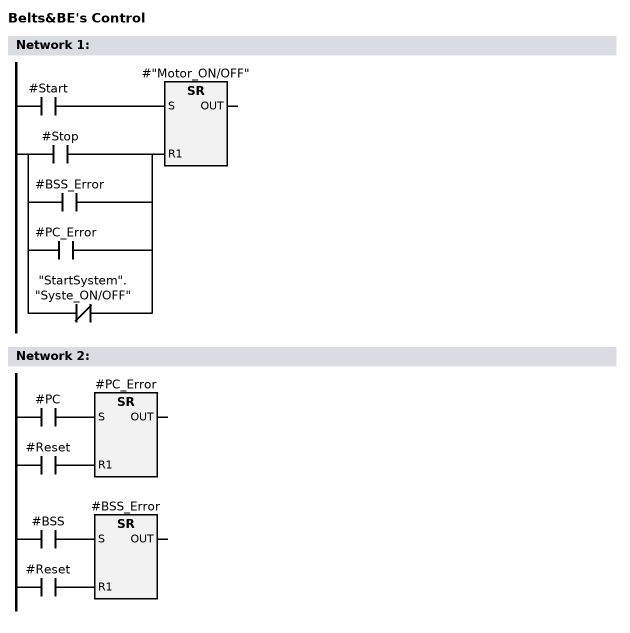
   RUNG wire#powerrail
      Contact( #Start )
      S_SR(operand := #"Motor_ON/OFF", r1 := wire#w1)
   END_RUNG
   RUNG wire#powerrail
      Contact( #Stop )
   END_RUNG wire#w1
   RUNG wire#powerrail
      Contact( #BSS_Error )
   END_RUNG wire#w1
   RUNG wire#powerrail
      Contact( #PC_Error )
   END_RUNG wire#w1
   RUNG wire#powerrail
      I_Contact( "StartSystem"."Syste_ON/OFF" )
   END_RUNG wire#w1
   // the same network as SCL:
   IF #Start THEN
       #"Motor_ON/OFF" := TRUE;   // SR flip-flop
   END_IF;
   IF #Stop OR #BSS_Error OR #PC_Error OR NOT "StartSystem"."Syste_ON/OFF" THEN
       #"Motor_ON/OFF" := FALSE;
   END_IF;
END_REGION

REGION Network 2
   RUNG wire#powerrail
      Contact( #PC )
      S_SR(operand := #PC_Error, r1 := wire#w1)
   END_RUNG
   RUNG wire#powerrail
      Contact( #Reset )
   END_RUNG wire#w1
   RUNG wire#powerrail
      Contact( #BSS )
      S_SR(operand := #BSS_Error, r1 := wire#w2)
   END_RUNG
   RUNG wire#powerrail
      Contact( #Reset )
   END_RUNG wire#w2
   // the same network as SCL:
   IF #PC THEN
       #PC_Error := TRUE;   // SR flip-flop
   END_IF;
   IF #Reset THEN #PC_Error := FALSE; END_IF;
   IF #BSS THEN
       #BSS_Error := TRUE;   // SR flip-flop
   END_IF;
   IF #Reset THEN #BSS_Error := FALSE; END_IF;
END_REGION
END_FUNCTION

FUNCTION "MotorDrives Control" : Void   // FC4, LAD
{ S7_Optimized_Access := 'TRUE' }
VERSION : 0.1
   VAR_INPUT
      Start : Bool;
      Stop : Bool;
   END_VAR
   VAR_IN_OUT
      "Motor_ON/OFF" : Bool;
   END_VAR
BEGIN

REGION Network 1
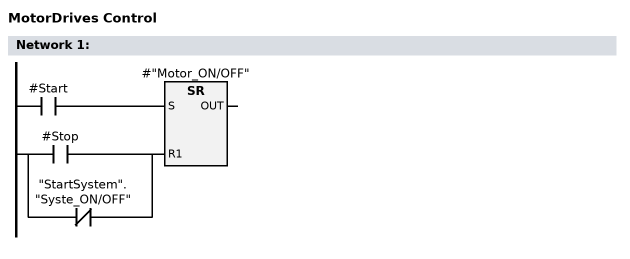
   RUNG wire#powerrail
      Contact( #Start )
      S_SR(operand := #"Motor_ON/OFF", r1 := wire#w1)
   END_RUNG
   RUNG wire#powerrail
      Contact( #Stop )
   END_RUNG wire#w1
   RUNG wire#powerrail
      I_Contact( "StartSystem"."Syste_ON/OFF" )
   END_RUNG wire#w1
   // the same network as SCL:
   IF #Start THEN
       #"Motor_ON/OFF" := TRUE;   // SR flip-flop
   END_IF;
   IF #Stop OR NOT "StartSystem"."Syste_ON/OFF" THEN #"Motor_ON/OFF" := FALSE; END_IF;
END_REGION
END_FUNCTION

FUNCTION "FowardRevers_Belts" : Void   // FC11, LAD
{ S7_Optimized_Access := 'TRUE' }
VERSION : 0.1
   VAR_INPUT
      Foward : Bool;
      Reverse : Bool;
      Stop : Bool;
      PC : Bool;
      BSS : Bool;
      Reset : Bool;
   END_VAR
   VAR_IN_OUT
      BSS_Error : Bool;
      PC_Error : Bool;
      Reverse_Mode : Bool;
      Foward_Mode : Bool;
   END_VAR
   VAR_TEMP
      Hold_On : Bool;
   END_VAR
BEGIN

REGION Network 1: Foward Mode
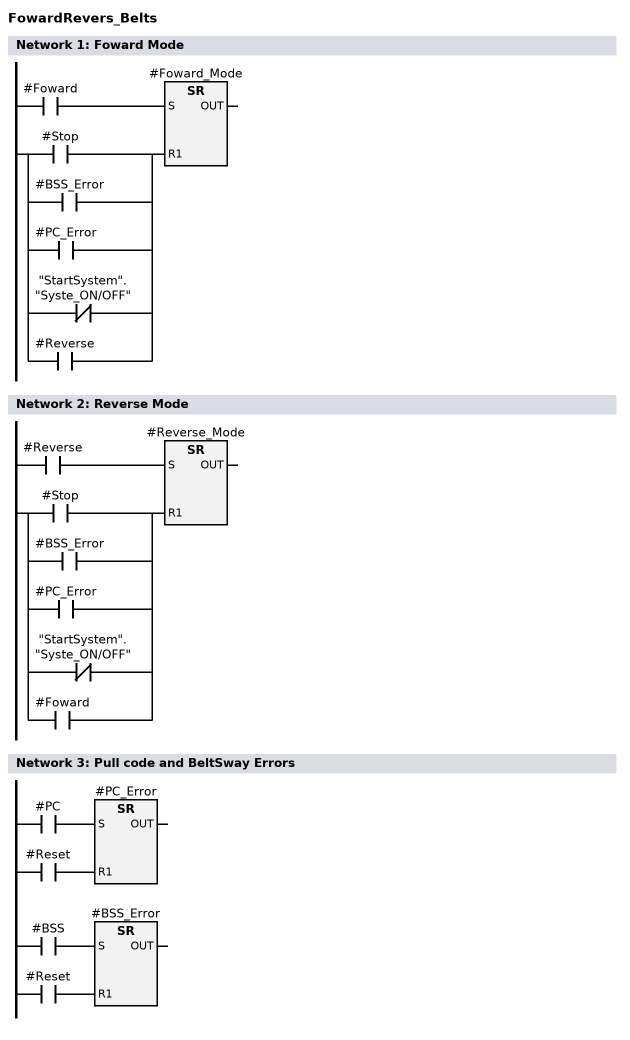
   RUNG wire#powerrail
      Contact( #Foward )
      S_SR(operand := #Foward_Mode, r1 := wire#w1)
   END_RUNG
   RUNG wire#powerrail
      Contact( #Stop )
   END_RUNG wire#w1
   RUNG wire#powerrail
      Contact( #BSS_Error )
   END_RUNG wire#w1
   RUNG wire#powerrail
      Contact( #PC_Error )
   END_RUNG wire#w1
   RUNG wire#powerrail
      I_Contact( "StartSystem"."Syste_ON/OFF" )
   END_RUNG wire#w1
   RUNG wire#powerrail
      Contact( #Reverse )
   END_RUNG wire#w1
   // the same network as SCL:
   IF #Foward THEN
       #Foward_Mode := TRUE;   // SR flip-flop
   END_IF;
   IF #Stop OR #BSS_Error OR #PC_Error OR NOT "StartSystem"."Syste_ON/OFF" OR #Reverse THEN
       #Foward_Mode := FALSE;
   END_IF;
END_REGION

REGION Network 2: Reverse Mode
   RUNG wire#powerrail
      Contact( #Reverse )
      S_SR(operand := #Reverse_Mode, r1 := wire#w1)
   END_RUNG
   RUNG wire#powerrail
      Contact( #Stop )
   END_RUNG wire#w1
   RUNG wire#powerrail
      Contact( #BSS_Error )
   END_RUNG wire#w1
   RUNG wire#powerrail
      Contact( #PC_Error )
   END_RUNG wire#w1
   RUNG wire#powerrail
      I_Contact( "StartSystem"."Syste_ON/OFF" )
   END_RUNG wire#w1
   RUNG wire#powerrail
      Contact( #Foward )
   END_RUNG wire#w1
   // the same network as SCL:
   IF #Reverse THEN
       #Reverse_Mode := TRUE;   // SR flip-flop
   END_IF;
   IF #Stop OR #BSS_Error OR #PC_Error OR NOT "StartSystem"."Syste_ON/OFF" OR #Foward THEN
       #Reverse_Mode := FALSE;
   END_IF;
END_REGION

REGION Network 3: Pull code and BeltSway Errors
   RUNG wire#powerrail
      Contact( #PC )
      S_SR(operand := #PC_Error, r1 := wire#w1)
   END_RUNG
   RUNG wire#powerrail
      Contact( #Reset )
   END_RUNG wire#w1
   RUNG wire#powerrail
      Contact( #BSS )
      S_SR(operand := #BSS_Error, r1 := wire#w2)
   END_RUNG
   RUNG wire#powerrail
      Contact( #Reset )
   END_RUNG wire#w2
   // the same network as SCL:
   IF #PC THEN
       #PC_Error := TRUE;   // SR flip-flop
   END_IF;
   IF #Reset THEN #PC_Error := FALSE; END_IF;
   IF #BSS THEN
       #BSS_Error := TRUE;   // SR flip-flop
   END_IF;
   IF #Reset THEN #BSS_Error := FALSE; END_IF;
END_REGION
END_FUNCTION

// folder: WeighFeeders(PID'S)

FUNCTION "LoadCell_Simulation(FC)" : Void   // FC2, LAD
{ S7_Optimized_Access := 'TRUE' }
VERSION : 0.1
   VAR_INPUT
      Max_tph : Real;
      "MotorSpeed%" : Real;
      SetPoint : Real;
   END_VAR
   VAR_IN_OUT
      LoadCell_Weight : Real;
   END_VAR
   VAR_TEMP
      Measured_Flow : Real;
      Measured_Outflow : Real;
      CurrentMeasured_Outflow : Real;
   END_VAR
BEGIN

REGION Network 1 (SCL): Max_tph is the maximum load a belt can carry in tons per hour.
   // The 0.0000278 is just 0.1sec(Cyclic interrup calling the function) divided by 3600 seconds(1 hour)
   // 2 Measured_Flows are the inflow and outflow of the belt. eg if inflow is 75t/h outflow is also 75t/h
   IF #SetPoint <> 0 THEN
       #Measured_Outflow := #SetPoint - 5;
       #CurrentMeasured_Outflow := 0.000278 * #Measured_Outflow;
       #Measured_Flow := 0.000278 * (#Max_tph / 100) * #"MotorSpeed%";
       #LoadCell_Weight := #LoadCell_Weight + #Measured_Flow - #CurrentMeasured_Outflow;
   END_IF;
END_REGION

REGION Network 2
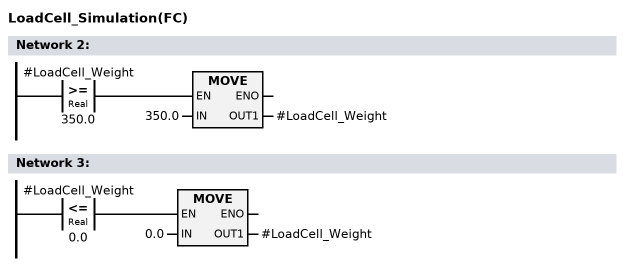
   RUNG wire#powerrail
      { S7_Templates := "SrcType := Real" } GE_Contact(in1 := #LoadCell_Weight, in2 := 350.0)
      Move(in := 350.0, out1 => #LoadCell_Weight)
   END_RUNG
   // the same network as SCL:
   IF #LoadCell_Weight >= 350.0 THEN #LoadCell_Weight := 350.0; END_IF;
END_REGION

REGION Network 3
   RUNG wire#powerrail
      { S7_Templates := "SrcType := Real" } LE_Contact(in1 := #LoadCell_Weight, in2 := 0.0)
      Move(in := 0.0, out1 => #LoadCell_Weight)
   END_RUNG
   // the same network as SCL:
   IF #LoadCell_Weight <= 0.0 THEN #LoadCell_Weight := 0.0; END_IF;
END_REGION
END_FUNCTION

FUNCTION "Setpoint Control" : Void   // FC6, LAD
{ S7_Optimized_Access := 'TRUE' }
VERSION : 0.1
   VAR_INPUT
      "WF_Setpoint%" : Real;
      Mill_TPH : Real;
   END_VAR
   VAR_OUTPUT
      Setpoint : Real;
   END_VAR
BEGIN

REGION Network 1 (SCL): Setpoint Calculation. Input percentage is calculated against the mill total TPH

   #Setpoint := (#"WF_Setpoint%" / 100.0) * #Mill_TPH;
END_REGION

REGION Network 2: Mill maximum TPH that can be set is 350
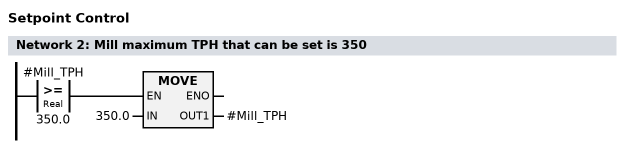
   RUNG wire#powerrail
      { S7_Templates := "SrcType := Real" } GE_Contact(in1 := #Mill_TPH, in2 := 350.0)
      Move(in := 350.0, out1 => #Mill_TPH)
   END_RUNG
   // the same network as SCL:
   IF #Mill_TPH >= 350.0 THEN #Mill_TPH := 350.0; END_IF;
END_REGION
END_FUNCTION

FUNCTION "Setpoint_MoveFunction" : Void   // FC9, LAD
{ S7_Optimized_Access := 'TRUE' }
VERSION : 0.1
   VAR_INPUT
      "Clinker%Setpoint" : Real;
      "Pozzo%Setpoint" : Real;
      "Gypsum%Setpoint" : Real;
      "Lime%Setpoint" : Real;
   END_VAR
   VAR_OUTPUT
      "WF_Clinker%Setpoint" : Real;
      "WF_Pozzo%Setpoint" : Real;
      "WF_Gypsum%Setpoint" : Real;
      "WF_Lime%Setpoint" : Real;
   END_VAR
BEGIN

REGION Network 1
